	//Step 37-38: Read DC bus voltage (S-0-0380)
	37: //Step 37: Trigger FB
		_CmdReadDcBusVoltage( Execute := FALSE, Axis := _Axis );
		_CmdReadDcBusVoltage( Execute := TRUE, Timeout := DEFAULT_ADS_TIMEOUT, Axis := _Axis );
		IF _CmdReadDcBusVoltage.Busy THEN _Step := 38; END_IF
		
	38: //Step 38: Check for errors and write to diagnostic parameter
		_CmdReadDcBusVoltage( Execute := FALSE, Axis := _Axis );
		IF NOT _CmdReadDcBusVoltage.Busy THEN
			IF NOT _CmdReadDcBusVoltage.Error THEN
				_DcBusVoltage	:= _CmdReadDcBusVoltage.DcBusVoltage;
			ELSE
				Error 			:= TRUE;
				ErrorStep		:= _Step;
				AdsErrId		:= _CmdReadDcBusVoltage.AdsErrId;
				SercosErrId		:= _CmdReadDcBusVoltage.SercosErrId;
			END_IF
			_Step := 39;
		END_IF
		
	//Step 39-40: Read actual main voltage (P-0-0200)
	39: //Step 39: Trigger FB
		_CmdReadMainVoltage( Execute := FALSE, Axis := _Axis );
		_CmdReadMainVoltage( Execute := TRUE, Timeout := DEFAULT_ADS_TIMEOUT, Axis := _Axis );
		IF _CmdReadMainVoltage.Busy THEN _Step := 40; END_IF
		
	40: //Step 40: Check for errors and write to diagnostic parameter
		_CmdReadMainVoltage( Execute := FALSE, Axis := _Axis );
		IF NOT _CmdReadMainVoltage.Busy THEN
			IF NOT _CmdReadMainVoltage.Error THEN
				_ActMainPeakVoltage	:= _CmdReadMainVoltage.ActualMainVoltage;
				_ActMainRMSVoltage	:= _ActMainPeakVoltage/(SQRT(2));	
			ELSE
				Error 				:= TRUE;
				ErrorStep			:= _Step;
				ErrorStep			:= _Step;
				AdsErrId			:= _CmdReadMainVoltage.AdsErrId;
				SercosErrId			:= _CmdReadMainVoltage.SercosErrId;
			END_IF	
			_Step := 41;		
		END_IF
		
	//Step 41-42: Read Safety State (P-0-2002) and set state bool	
	41: //Step 41: Trigger FB
		_CmdSoERead( Execute := FALSE, Axis :=_Axis);	
		_CmdSoERead( Execute := TRUE, Idn := P_0_IDN + 2002, Element :=16#40, pDstBuf :=ADR(_SafetyOptionState), BufLen :=SIZEOF(_SafetyOptionState), Timeout := DEFAULT_ADS_TIMEOUT, Axis := _Axis);
		IF _CmdSoERead.Busy THEN _Step := 42; END_IF
		
	42: //Step 42: Check for errors and write to field parameter
		_CmdSoERead(Execute:= FALSE, Axis := _Axis);
		IF NOT _CmdSoERead.Busy THEN	
			IF NOT _CmdSoERead.Error THEN
				_SafetyStateBool	:= _SafetyOptionState.0;
			ELSE
				Error				:= TRUE;
				ErrorStep			:= _Step;
				AdsErrId			:= _CmdSoERead.AdsErrId;
				SercosErrId			:= _CmdSoERead.SercosErrId;
			END_IF
			_Step := 43;
		END_IF
	
	//Step 43-44: Read torque peak (P-0-0094)	
	43: //Step 43: Trigger FB
		_CmdSoERead( Execute := FALSE, Axis :=_Axis);	
		_CmdSoERead( Execute := TRUE, Idn := P_0_IDN + 92, Element :=16#40, pDstBuf :=ADR(_TorquePeak), BufLen :=SIZEOF(_TorquePeak), Timeout := DEFAULT_ADS_TIMEOUT, Axis := _Axis);
		IF _CmdSoERead.Busy THEN _Step := 44; END_IF
		
	44: //Step 44: Check for errors and write to field parameter
		_CmdSoERead(Execute:= FALSE, Axis := _Axis);
		IF NOT _CmdSoERead.Busy THEN	
			IF NOT _CmdSoERead.Error THEN
				;
			ELSE
				Error			:= TRUE;
				ErrorStep		:= _Step;
				AdsErrId		:= _CmdSoERead.AdsErrId;
				SercosErrId		:= _CmdSoERead.SercosErrId;
			END_IF
			_Step := 45;
		END_IF
		
	//Step 45-46: Read torque feedback percentage (S-0-0084)	
	45: //Step 45: Trigger FB	
		_CmdSoERead( Execute := FALSE, Axis :=_Axis);	
		_CmdSoERead( Execute := TRUE, Idn := S_0_IDNs + 84, Element :=16#40, pDstBuf :=ADR(_TorqueFeedbackPercent), BufLen :=SIZEOF(_TorqueFeedbackPercent), Timeout := DEFAULT_ADS_TIMEOUT, Axis := _Axis);
		IF _CmdSoERead.Busy THEN _Step := 46; END_IF
		
	46: //Step 46: Check for errors and write to field parameter after converting percentage of peak into current Nm
		//Note: In drive manager value read for parameter is real, when read in code however the value returned is an int. i.e. Torque peak - in DM = 6.0, returned from SOE read 6000, Torque % - in DM = 6.7 returned 67. (check date size in IDN description manual for 16 bit or 23 bit size.
		_CmdSoERead(Execute:= FALSE, Axis := _Axis);
		IF NOT _CmdSoERead.Busy THEN	
			IF NOT _CmdSoERead.Error THEN 
				_TorqueFeedback := (INT_TO_REAL(_TorqueFeedbackPercent)/10)*(DINT_TO_LREAL(_TorquePeak)/100000);
			ELSE
				Error			:= TRUE;
				ErrorStep		:= _Step;
				AdsErrId		:= _CmdSoERead.AdsErrId;
				SercosErrId		:= _CmdSoERead.SercosErrId;
			END_IF
			_Step := 47;
		END_IF

	//Step 47-48: Read motor break current (P-0-0064)
	47: //Step 37: Trigger FB
		_CmdSoERead( Execute := FALSE, Axis :=_Axis);	
		_CmdSoERead( Execute := TRUE, Idn := P_0_IDN + 64, Element :=16#40, pDstBuf :=ADR(_ActMotorBreakCurrentRead), BufLen :=SIZEOF(_ActMotorBreakCurrentRead), Timeout := DEFAULT_ADS_TIMEOUT, Axis := _Axis);
		IF _CmdSoERead.Busy THEN _Step := 48; END_IF
		
	48: //Step 48: Check for errors and write to status parameter
		_CmdSoERead(Execute:= FALSE, Axis := _Axis);
		IF NOT _CmdSoERead.Busy THEN	
			IF NOT _CmdSoERead.Error THEN
				_ActMotorBreakCurrent := INT_TO_REAL(_ActMotorBreakCurrentRead)/1000;
			ELSE
				Error			:= TRUE;
				ErrorStep		:= _Step;
				AdsErrId		:= _CmdSoERead.AdsErrId;
				SercosErrId		:= _CmdSoERead.SercosErrId;
			END_IF
			_Step := 49;	
		END_IF
	
	49: //Step 49: Calulate normal torque limit from peak
		_NormalTorqueLimitNm := (UINT_TO_REAL(_NormalTorqueLimit)/100) * (DINT_TO_LREAL(_TorquePeak)/1000);
		_Step := 50;
	
	// Step 50-51: Get motor peak force (P-0-0128)
	50: //Step 50: Trigger FB
		_CmdSoERead( Execute := FALSE, Axis :=_Axis);	
		_CmdSoERead( Execute := TRUE, Idn := P_0_IDN + 128, Element :=16#40, pDstBuf :=ADR(_MotorPeakForceRead), BufLen :=SIZEOF(_MotorPeakForceRead), Timeout := DEFAULT_ADS_TIMEOUT, Axis := _Axis);
		IF _CmdSoERead.Busy THEN _Step := 51; END_IF
		
	51: //Step 48: Check for errors and write to status parameter
		_CmdSoERead(Execute:= FALSE, Axis := _Axis);
		IF NOT _CmdSoERead.Busy THEN	
			IF NOT _CmdSoERead.Error THEN
				_MotorPeakForce := UINT_TO_REAL(_MotorPeakForceRead)/1000;
			ELSE
				Error			:= TRUE;
				ErrorStep		:= _Step;
				AdsErrId		:= _CmdSoERead.AdsErrId;
				SercosErrId		:= _CmdSoERead.SercosErrId;
			END_IF
			_Step		:= 0;	
		END_IF
		
	52: //Display diagnostics function error
		IF Error THEN
			;
		END_IF
END_CASE
END_METHOD

METHOD PRIVATE M_Homing
VAR_INPUT
END_VAR
VAR_INST
             	                			
	_HomingJogPos						: BOOL;	
	{attribute 'tc_no_symbol'}                	                			
	_CMD_Home							: MC_HOME;
	{attribute 'tc_no_symbol'}                	                			
	_CMD_SetPosition					: MC_SETPOSITION;
	{attribute 'tc_no_symbol'}                	                			
	_CMD_SoEAX5000SetPositionOffset		: FB_SoEAX5000SetPositionOffset;
	{attribute 'tc_no_symbol'}   
	_SoEAX5000SetPositionOffsetBusyLatch: BOOL;								//Due to no done bit for function this bit latched on busy then for use in detecting falling edge
	{attribute 'tc_no_symbol'}                	                			
	_CMD_SoEAX5000DeletePositionOffset	: FB_SoEAX5000DeletePositionOffset;
	{attribute 'tc_no_symbol'}                	                				
	_CMD_HomeJOG						: MC_JOG;
	{attribute 'tc_no_symbol'}                	                			
	_R_Trig								: ARRAY[0..6] OF R_TRIG;
END_VAR
// ----------------------------------------
// Homing Outputs
// ----------------------------------------
_HomingEN:=_CMD_Home.Busy OR _CMD_SetPosition.Busy OR _CMD_SoEAX5000SetPositionOffset.Busy;
IF _CMD_Home.Busy OR _CMD_SetPosition.Busy OR _CMD_SoEAX5000SetPositionOffset.Busy THEN _Homed := FALSE; END_IF
IF _CMD_Home.Done OR _CMD_SetPosition.Done OR _R_Trig[1].Q THEN _Homed := TRUE;_SoEAX5000SetPositionOffsetBusyLatch:=FALSE; END_IF

// ----------------------------------------
// Error Handler	
// ----------------------------------------
_r_Trig[0](clk :=
(_CMD_Home.Execute AND _CMD_Home.Error) OR 
(_CMD_SetPosition.Execute AND _CMD_SetPosition.Error) OR
(_CMD_SoEAX5000DeletePositionOffset.Execute AND _CMD_SoEAX5000DeletePositionOffset.Error) OR
(_CMD_SoEAX5000SetPositionOffset.Execute AND _CMD_SoEAX5000SetPositionOffset.Error));


// ----------------------------------------
// Manual Home Selection	
// ----------------------------------------
IF _ManHome.Select AND NOT _ManHome.Interlock THEN
	_ManHome.Select :=TRUE;
ELSE
	_ManHome.Select :=FALSE;
END_IF

IF ((_HomeMode < 3) AND NOT Control.PackMLState.Stopped AND NOT Control.PackMLState.Idle)  THEN
	_ManHome.Messages:= 'Axis Cannot be homed.$LSystem is not in an Stopped or Idle State.';
ELSIF((_HomeMode >= 3) AND NOT Control.PackMLState.Aborted) THEN
	_ManHome.Messages:= 'Axis Cannot be homed as the Machine is not De-energized.$LSystem is not in an Aborted State';
ELSIF _r_Trig[0].Q THEN
	_ManHome.Messages:= 'Axis Homing Error Occurred';
ELSE
	IF (_HomeMode < 3) THEN
		_ManHome.Messages:= 'Axis Ready to be Homed.$LThis will cause motion towards the Switch.';
	ELSE
		_ManHome.Messages:= 'Axis Ready to be Homed.$LThe Axis will remain stationary.';
	END_IF
END_IF


IF _CMD_Home.Done OR _CMD_SetPosition.Done OR _R_Trig[1].Q
	OR ((_HomeMode < 3) AND NOT Control.PackMLState.Stopped AND NOT Control.PackMLState.Idle)
	OR ((_HomeMode >= 3) AND NOT Control.PackMLState.Aborted)
	OR _r_Trig[0].Q THEN
	_ManHome.Interlock :=TRUE; 
ELSE
	_ManHome.Interlock :=FALSE;
END_IF


IF _ManHome.Select  THEN
	_ManHome.Queued :=TRUE;
	_ManHome.Messages:= 'Axis Homing Queued.';
ELSE
	_ManHome.Queued :=FALSE;
END_IF

IF _ManHome.Queued  THEN
	_ManHome.Messages:= 'Axis Homing in Progress.';
	_ManHome.Enabled :=TRUE;
ELSE
	_ManHome.Enabled :=FALSE;
END_IF

// ----------------------------------------
// MC Home	
// ----------------------------------------	
_CMD_Home(
	Axis:= _Axis, 
	Execute:= (_AutoHome OR _ManHome.Enabled) AND _HomeMode <=2,
	HomingMode:= MC_DefaultHoming, 
	BufferMode:= , 
	Options:= , 
	bCalibrationCam:= HomingInput, 
	Done=> , 
	Busy=> , 
	Active=> , 
	CommandAborted=> , 
	Error=> , 
	ErrorID=> );
_R_Trig[3](CLK:=_CMD_Home.Error);IF _R_Trig[3].Q THEN _AlarmNum := _CMD_Home.ErrorID; END_IF	

// ----------------------------------------
// MC Set Position	
// ----------------------------------------			
_CMD_SetPosition(
	Axis:= _Axis, 
	Execute:= (_AutoHome OR _ManHome.Enabled) AND _HomeMode = 3, 
	Position:= _PosMoveHome.Position, 
	Mode:= FALSE, 
	Options:= , 
	Done=> , 
	Busy=> , 
	Error=> , 
	ErrorID=> );	
_R_Trig[4](CLK:=_CMD_SetPosition.Error);IF _R_Trig[4].Q THEN _AlarmNum := _CMD_SetPosition.ErrorID; END_IF	

// ----------------------------------------
// MC Set Position Offset	
// ----------------------------------------		
//* Note to Set P-0-0275 = 2.Use Drive Memory	
_CMD_SoEAX5000SetPositionOffset(
	Execute:= (_AutoHome OR _ManHome.Enabled) AND _HomeMode = 4, 
	Position:= _PosMoveHome.Position, 
	Relative:= FALSE, 
	Feedback:= tc2_mc2_Drive.E_PositionOffsetFeedback.ePositionOffsetFeedback1, 
	Memory:=  tc2_mc2_Drive.E_PositionOffsetMemory.ePositionOffsetMemory_Drive, 
	Busy=> , 
	Error=> , 
	ErrorID=> , 
	Axis:= _Axis);
_R_Trig[5](CLK:=_CMD_SoEAX5000SetPositionOffset.Error);IF _R_Trig[5].Q THEN _AlarmNum := _CMD_SoEAX5000SetPositionOffset.ErrorID; END_IF
IF _CMD_SoEAX5000SetPositionOffset.Busy THEN _SoEAX5000SetPositionOffsetBusyLatch := TRUE; END_IF
_R_Trig[1](CLK:=_SoEAX5000SetPositionOffsetBusyLatch AND NOT _CMD_SoEAX5000SetPositionOffset.Busy);
END_METHOD

METHOD PRIVATE M_Jogging
VAR_INPUT
END_VAR
VAR_INST
	{attribute 'tc_no_symbol'}                	                			
	_accelRate							: LREAL;
	{attribute 'tc_no_symbol'}                	                			
	_decelRate							: LREAL;
	{attribute 'tc_no_symbol'}                	                			
	_jerkTime							: LREAL;
	{attribute 'tc_no_symbol'}                	                			
	_jerkValue							: LREAL;
	{attribute 'tc_no_symbol'}                	                			
	_enableJog							: BOOL;
	{attribute 'tc_no_symbol'}                	                			
	_enableManPos						: BOOL;
	{attribute 'tc_no_symbol'}                	                			
	_manPosAbsActive					: BOOL;
	{attribute 'tc_no_symbol'}                	                			
	_manPosModActive					: BOOL;
	{attribute 'tc_no_symbol'}                	                			
	_manPosRelActive					: BOOL;
	{attribute 'tc_no_symbol'}                	                			
	_CMD_JOG							: MC_JOG;
	{attribute 'tc_no_symbol'}                	                			
	_CMD_MovePosManAbs					: MC_MOVEABSOLUTE;
	{attribute 'tc_no_symbol'}                	                			
	_CMD_MovePosManMod					: MC_MOVEMODULO;
	{attribute 'tc_no_symbol'}                	                			
	_CMD_MovePosManRel					: MC_MOVERELATIVE;
	{attribute 'tc_no_symbol'}                	                			
	_CMD_ManMoveHalt					: MC_HALT;
END_VAR
VAR_INST // added by the converter: edge detectors and wires of the graphical bodies
    _w1, _w2 : BOOL;
    _rt1, _rt2, _rt3, _rt4, _rt5 : R_TRIG;
END_VAR
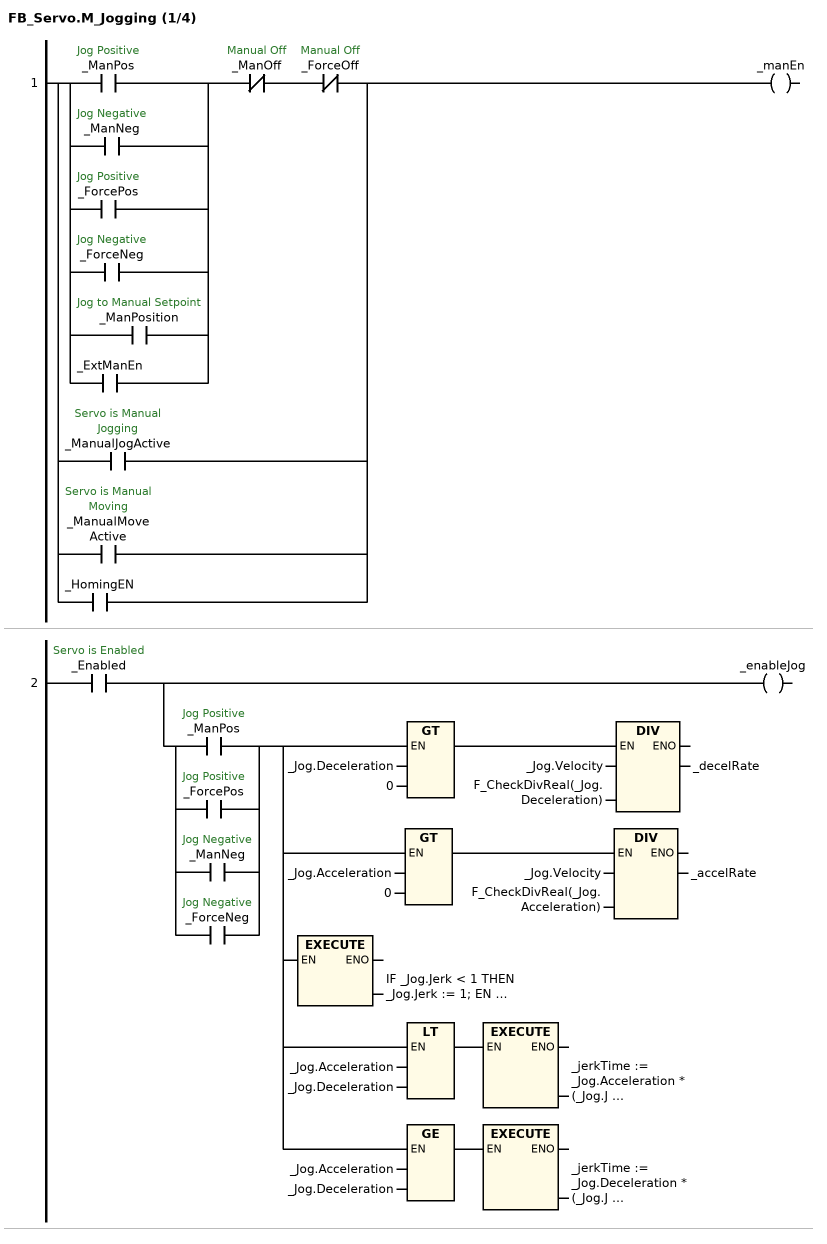
// NETWORK 1
//   _ManPos: Jog Positive
//   _ManNeg: Jog Negative
//   _ForcePos: Jog Positive
//   _ForceNeg: Jog Negative
//   _ManPosition: Jog to Manual Setpoint
//   _ManOff: Manual Off
//   _ForceOff: Manual Off
//   _ManualJogActive: Servo is Manual Jogging
//   _ManualMoveActive: Servo is Manual Moving
_manEn := (_ManPos OR _ManNeg OR _ForcePos OR _ForceNeg OR _ManPosition OR _ExtManEn) AND NOT _ManOff AND NOT _ForceOff OR _ManualJogActive OR _ManualMoveActive OR _HomingEN;

// NETWORK 2
//   _Enabled: Servo is Enabled
//   _ManPos: Jog Positive
//   _ForcePos: Jog Positive
//   _ManNeg: Jog Negative
//   _ForceNeg: Jog Negative
//   _Jog.Velocity: Velocity Value of Move
//   F_CheckDivReal(_Jog.Deceleration): Deceleration Value of Move
//   F_CheckDivReal(_Jog.Acceleration): Accleration Value of Move
//   _Jog.Acceleration: Accleration Value of Move
//   _Jog.Deceleration: Deceleration Value of Move
_enableJog := _Enabled;
_w1 := _Enabled AND (_ManPos OR _ForcePos OR _ManNeg OR _ForceNeg);
IF _w1 AND _Jog.Deceleration > 0 THEN _decelRate := _Jog.Velocity / (F_CheckDivReal(_Jog.Deceleration)); END_IF
IF _w1 AND _Jog.Acceleration > 0 THEN _accelRate := _Jog.Velocity / (F_CheckDivReal(_Jog.Acceleration)); END_IF
IF _w1 THEN
    IF _Jog.Jerk < 1 THEN _Jog.Jerk := 1; END_IF
    IF _Jog.Jerk > 100 THEN _Jog.Jerk := 100; END_IF
END_IF
IF _w1 AND _Jog.Acceleration < _Jog.Deceleration THEN
    _jerkTime := _Jog.Acceleration * (_Jog.Jerk / 100);
    IF _jerkTime > 0 THEN
    	_jerkValue := _accelRate / F_CheckDivReal(LREAL_TO_REAL(_jerkTime));
    END_IF
END_IF
IF _w1 AND _Jog.Acceleration >= _Jog.Deceleration THEN
    _jerkTime := _Jog.Deceleration * (_Jog.Jerk / 100);
    IF _jerkTime > 0 THEN
    	_jerkValue := _decelRate / F_CheckDivReal(LREAL_TO_REAL(_jerkTime));
    END_IF
END_IF

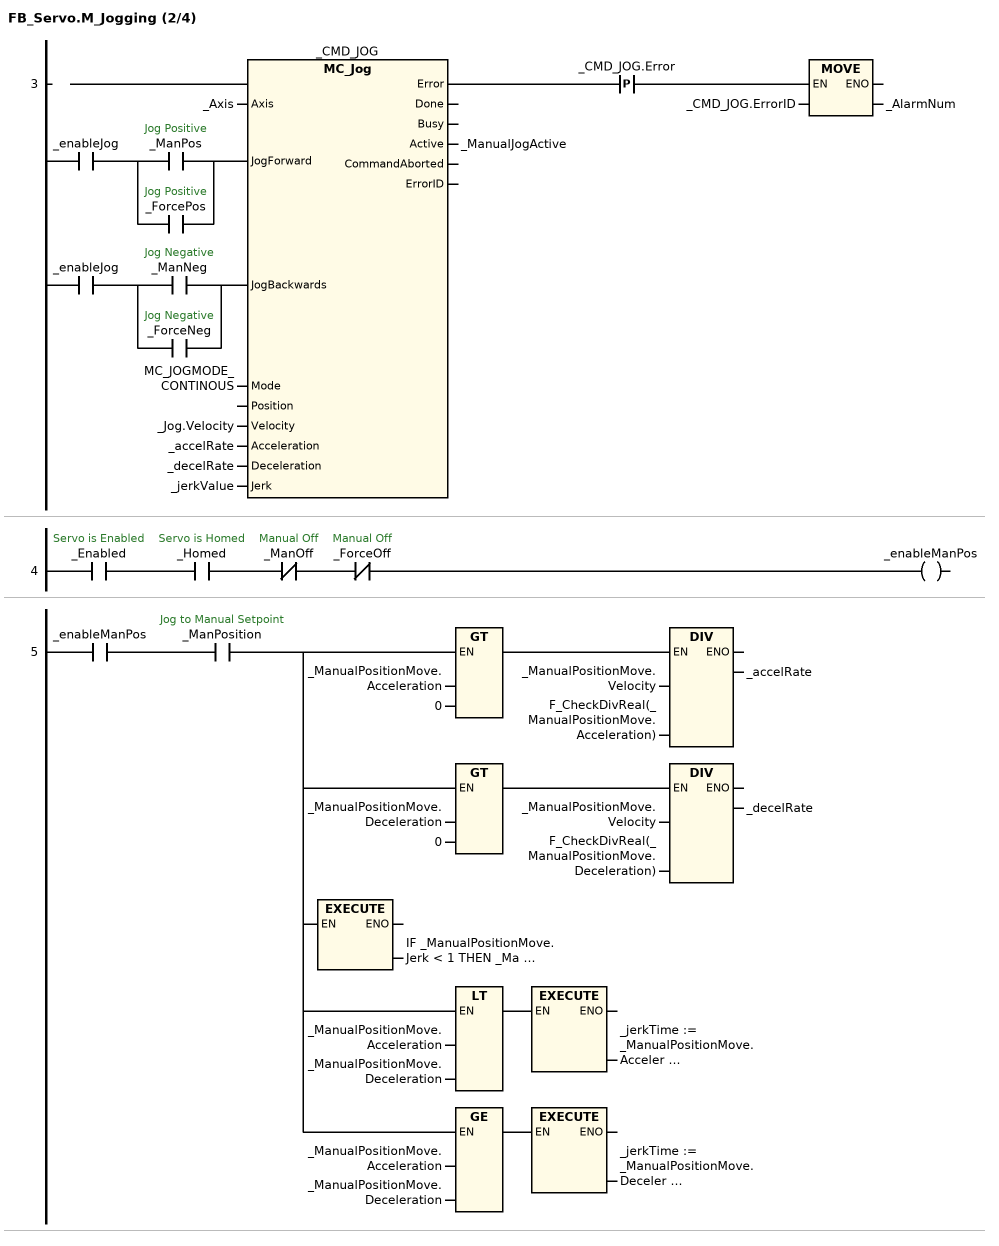
// NETWORK 3
//   _ManPos: Jog Positive
//   _ForcePos: Jog Positive
//   _ManNeg: Jog Negative
//   _ForceNeg: Jog Negative
//   MC_JOGMODE_CONTINOUS: axis moves as long as the jog button is pressed using parameterized dynamics
//   _Jog.Velocity: Velocity Value of Move
//   _ManualJogActive: Servo is Manual Jogging
_CMD_JOG(
    Axis := _Axis,
    JogForward := _enableJog AND (_ManPos OR _ForcePos),
    JogBackwards := _enableJog AND (_ManNeg OR _ForceNeg),
    Mode := MC_JOGMODE_CONTINOUS,
    Velocity := _Jog.Velocity,
    Acceleration := _accelRate,
    Deceleration := _decelRate,
    Jerk := _jerkValue,
    Active => _ManualJogActive); // MC_Jog
_rt1(CLK := _CMD_JOG.Error);
IF _CMD_JOG.Error AND _rt1.Q THEN _AlarmNum := _CMD_JOG.ErrorID; END_IF

// NETWORK 4
//   _Enabled: Servo is Enabled
//   _Homed: Servo is Homed
//   _ManOff: Manual Off
//   _ForceOff: Manual Off
_enableManPos := _Enabled AND _Homed AND NOT _ManOff AND NOT _ForceOff;

// NETWORK 5
//   _ManPosition: Jog to Manual Setpoint
//   _ManualPositionMove.Velocity: Velocity Value of Move
//   F_CheckDivReal(_ManualPositionMove.Acceleration): Accleration Value of Move
//   F_CheckDivReal(_ManualPositionMove.Deceleration): Deceleration Value of Move
//   _ManualPositionMove.Acceleration: Accleration Value of Move
//   _ManualPositionMove.Deceleration: Deceleration Value of Move
_w2 := _enableManPos AND _ManPosition;
IF _w2 AND _ManualPositionMove.Acceleration > 0 THEN
    _accelRate := _ManualPositionMove.Velocity / (F_CheckDivReal(_ManualPositionMove.Acceleration));
END_IF
IF _w2 AND _ManualPositionMove.Deceleration > 0 THEN
    _decelRate := _ManualPositionMove.Velocity / (F_CheckDivReal(_ManualPositionMove.Deceleration));
END_IF
IF _w2 THEN
    IF _ManualPositionMove.Jerk < 1 THEN _ManualPositionMove.Jerk := 1; END_IF
    IF _ManualPositionMove.Jerk > 100 THEN _ManualPositionMove.Jerk := 100; END_IF
END_IF
IF _w2 AND _ManualPositionMove.Acceleration < _ManualPositionMove.Deceleration THEN
    _jerkTime := _ManualPositionMove.Acceleration * (_ManualPositionMove.Jerk / 100);
    IF _jerkTime > 0 THEN
    	_jerkValue := _accelRate / F_CheckDivReal(LREAL_TO_REAL(_jerkTime));
    END_IF
END_IF
IF _w2 AND _ManualPositionMove.Acceleration >= _ManualPositionMove.Deceleration THEN
    _jerkTime := _ManualPositionMove.Deceleration * (_ManualPositionMove.Jerk / 100);
    IF _jerkTime > 0 THEN
    	_jerkValue := _decelRate / F_CheckDivReal(LREAL_TO_REAL(_jerkTime));
    END_IF
END_IF

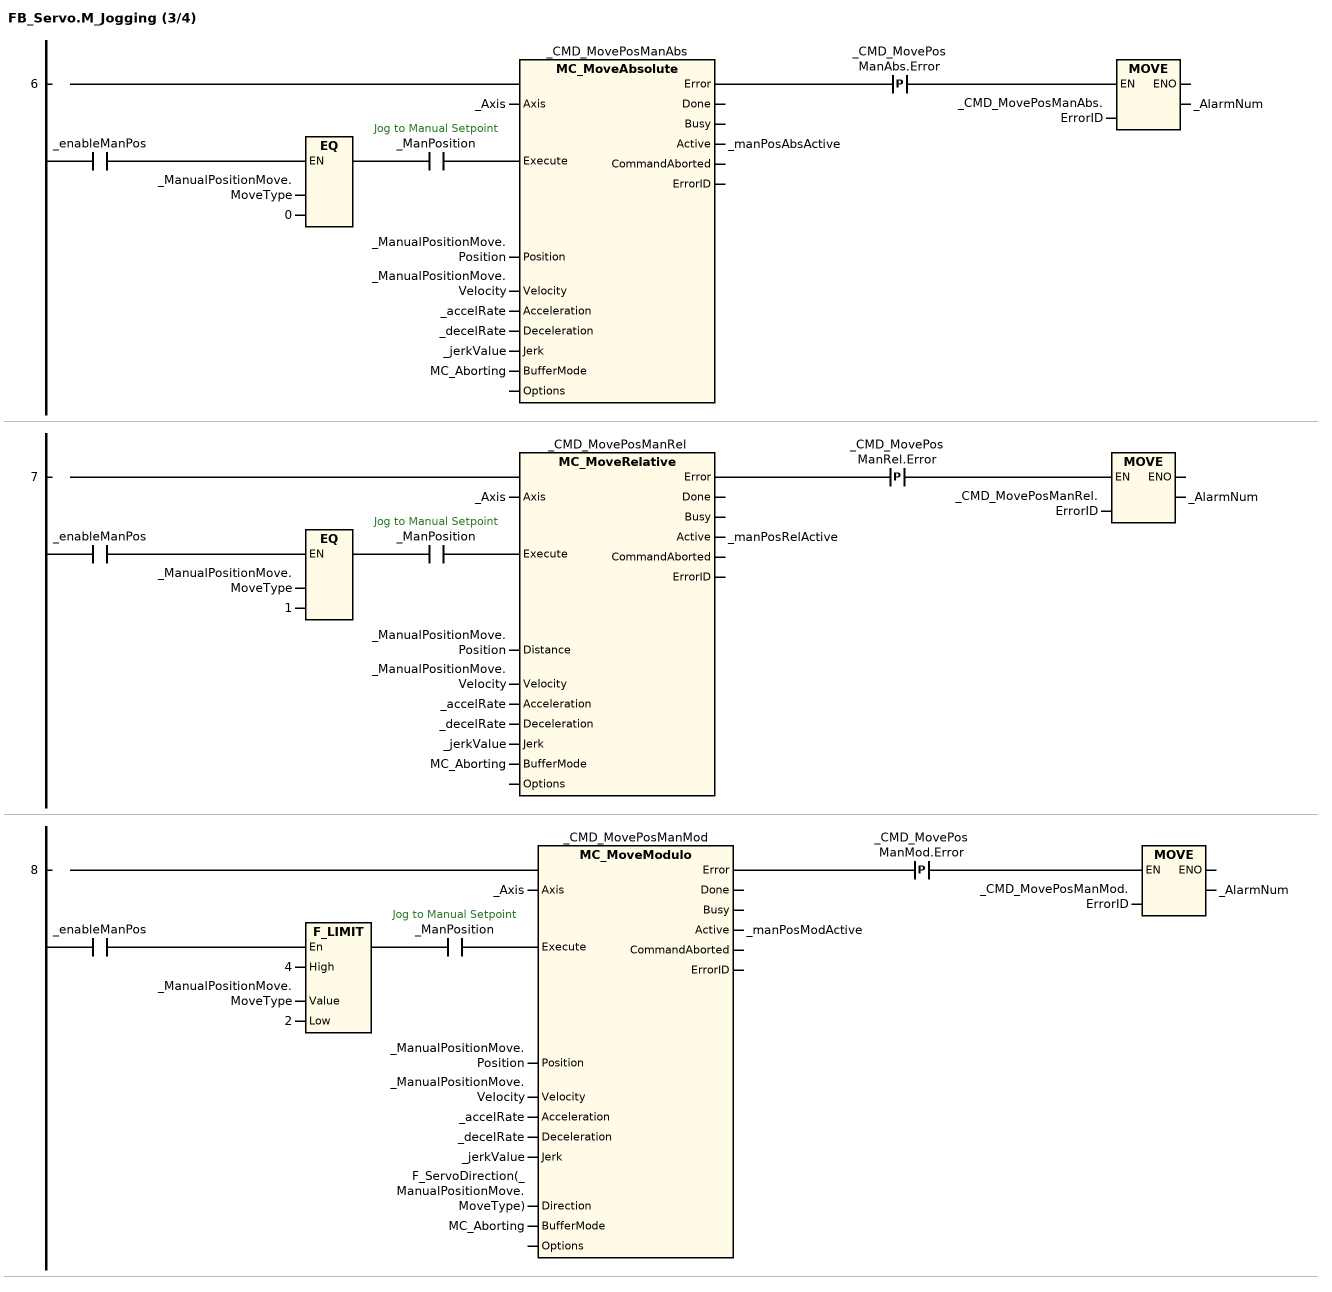
// NETWORK 6
//   _ManualPositionMove.MoveType: Move Type Configuration of Positional Move
//   _ManPosition: Jog to Manual Setpoint
//   _ManualPositionMove.Position: Position Value to Move to
//   _ManualPositionMove.Velocity: Velocity Value of Move
_CMD_MovePosManAbs(
    Axis := _Axis,
    Execute := (_enableManPos AND _ManualPositionMove.MoveType = 0) AND _ManPosition,
    Position := _ManualPositionMove.Position,
    Velocity := _ManualPositionMove.Velocity,
    Acceleration := _accelRate,
    Deceleration := _decelRate,
    Jerk := _jerkValue,
    BufferMode := MC_Aborting,
    Active => _manPosAbsActive); // MC_MoveAbsolute
_rt2(CLK := _CMD_MovePosManAbs.Error);
IF _CMD_MovePosManAbs.Error AND _rt2.Q THEN _AlarmNum := _CMD_MovePosManAbs.ErrorID; END_IF

// NETWORK 7
//   _ManualPositionMove.MoveType: Move Type Configuration of Positional Move
//   _ManPosition: Jog to Manual Setpoint
//   _ManualPositionMove.Position: Position Value to Move to
//   _ManualPositionMove.Velocity: Velocity Value of Move
_CMD_MovePosManRel(
    Axis := _Axis,
    Execute := (_enableManPos AND _ManualPositionMove.MoveType = 1) AND _ManPosition,
    Distance := _ManualPositionMove.Position,
    Velocity := _ManualPositionMove.Velocity,
    Acceleration := _accelRate,
    Deceleration := _decelRate,
    Jerk := _jerkValue,
    BufferMode := MC_Aborting,
    Active => _manPosRelActive); // MC_MoveRelative
_rt3(CLK := _CMD_MovePosManRel.Error);
IF _CMD_MovePosManRel.Error AND _rt3.Q THEN _AlarmNum := _CMD_MovePosManRel.ErrorID; END_IF

// NETWORK 8
//   _ManualPositionMove.MoveType: Move Type Configuration of Positional Move
//   _ManPosition: Jog to Manual Setpoint
//   _ManualPositionMove.Position: Position Value to Move to
//   _ManualPositionMove.Velocity: Velocity Value of Move
_CMD_MovePosManMod(
    Axis := _Axis,
    Execute := F_LIMIT(En := _enableManPos, High := 4, Value := _ManualPositionMove.MoveType, Low := 2) AND _ManPosition,
    Position := _ManualPositionMove.Position,
    Velocity := _ManualPositionMove.Velocity,
    Acceleration := _accelRate,
    Deceleration := _decelRate,
    Jerk := _jerkValue,
    Direction := F_ServoDirection(_ManualPositionMove.MoveType),
    BufferMode := MC_Aborting,
    Active => _manPosModActive); // MC_MoveModulo
_rt4(CLK := _CMD_MovePosManMod.Error);
IF _CMD_MovePosManMod.Error AND _rt4.Q THEN _AlarmNum := _CMD_MovePosManMod.ErrorID; END_IF

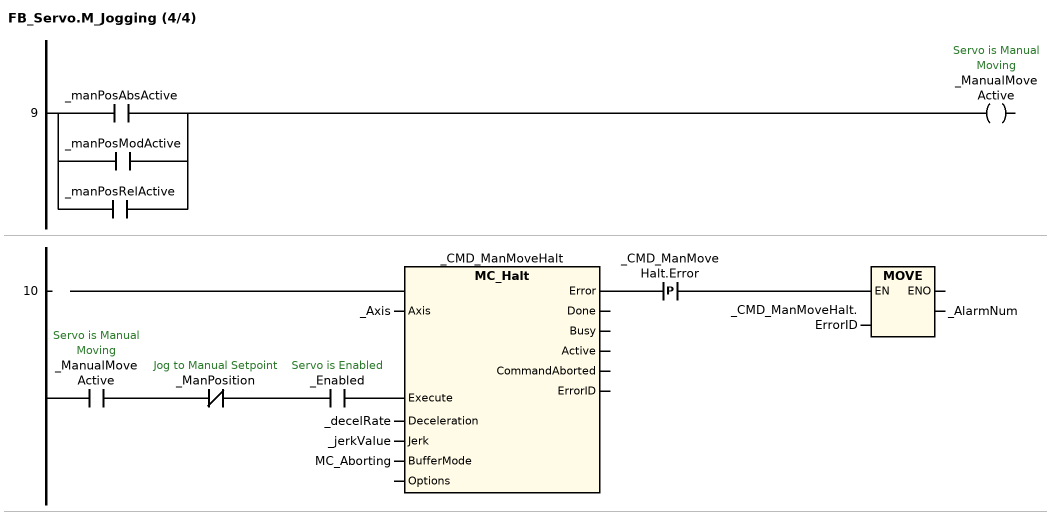
// NETWORK 9
//   _ManualMoveActive: Servo is Manual Moving
_ManualMoveActive := _manPosAbsActive OR _manPosModActive OR _manPosRelActive;

// NETWORK 10
//   _ManualMoveActive: Servo is Manual Moving
//   _ManPosition: Jog to Manual Setpoint
//   _Enabled: Servo is Enabled
_CMD_ManMoveHalt(
    Axis := _Axis,
    Execute := _ManualMoveActive AND NOT _ManPosition AND _Enabled,
    Deceleration := _decelRate,
    Jerk := _jerkValue,
    BufferMode := MC_Aborting); // MC_Halt
_rt5(CLK := _CMD_ManMoveHalt.Error);
IF _CMD_ManMoveHalt.Error AND _rt5.Q THEN _AlarmNum := _CMD_ManMoveHalt.ErrorID; END_IF
END_METHOD

METHOD PRIVATE M_MotionDynamicMove
VAR_INPUT
END_VAR
VAR_INST
	{attribute 'tc_no_symbol'}                	                			
	_fb_MovePosDynamic			: ARRAY [1..4] OF FB_ServoMotionDynamics;
	{attribute 'tc_no_symbol'}                	                			
	_enableDynamicMove			: BOOL;
	{attribute 'tc_no_symbol'}                	                			
	_Pos2MoveStart				: ST_MovePosition_SP;
	{attribute 'tc_no_symbol'}                	                			
	_CMD_MoveDynamicAbsStart	: ARRAY[1..4] OF MC_MOVEABSOLUTE;
	{attribute 'tc_no_symbol'}                	                			
	_CMD_MoveDynamicAbsEnd		: ARRAY[1..4] OF MC_MOVEABSOLUTE;
END_VAR
VAR_INST // added by the converter: edge detectors and wires of the graphical bodies
    _rt1, _rt2, _rt3, _rt4, _rt5, _rt6, _rt7, _rt8, _rt9, _rt10 : R_TRIG;
    _w1, _w2 : BOOL;
END_VAR
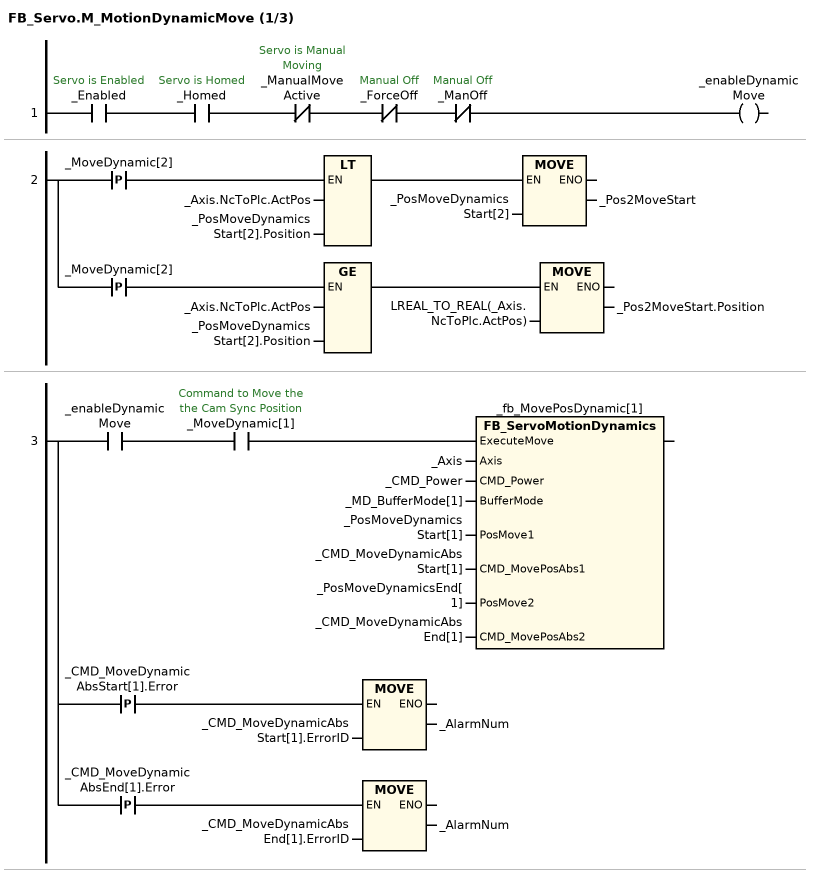
// NETWORK 1
//   _Enabled: Servo is Enabled
//   _Homed: Servo is Homed
//   _ManualMoveActive: Servo is Manual Moving
//   _ForceOff: Manual Off
//   _ManOff: Manual Off
_enableDynamicMove := _Enabled AND _Homed AND NOT _ManualMoveActive AND NOT _ForceOff AND NOT _ManOff;

// NETWORK 2
_rt1(CLK := _MoveDynamic[2]);
_w1 := _rt1.Q AND _Axis.NcToPlc.ActPos < _PosMoveDynamicsStart[2].Position;
IF _w1 THEN _Pos2MoveStart := _PosMoveDynamicsStart[2]; END_IF
_rt2(CLK := _MoveDynamic[2]);
_w2 := _rt2.Q AND _Axis.NcToPlc.ActPos >= _PosMoveDynamicsStart[2].Position;
IF _w2 THEN _Pos2MoveStart.Position := LREAL_TO_REAL(_Axis.NcToPlc.ActPos); END_IF

// NETWORK 3
//   _MoveDynamic[1]: Command to Move the the Cam Sync Position
_fb_MovePosDynamic[1](
    ExecuteMove := _enableDynamicMove AND _MoveDynamic[1],
    Axis := _Axis,
    CMD_Power := _CMD_Power,
    BufferMode := _MD_BufferMode[1],
    PosMove1 := _PosMoveDynamicsStart[1],
    CMD_MovePosAbs1 := _CMD_MoveDynamicAbsStart[1],
    PosMove2 := _PosMoveDynamicsEnd[1],
    CMD_MovePosAbs2 := _CMD_MoveDynamicAbsEnd[1]); // FB_ServoMotionDynamics
_rt3(CLK := _CMD_MoveDynamicAbsStart[1].Error);
IF _rt3.Q THEN _AlarmNum := _CMD_MoveDynamicAbsStart[1].ErrorID; END_IF
_rt4(CLK := _CMD_MoveDynamicAbsEnd[1].Error);
IF _rt4.Q THEN _AlarmNum := _CMD_MoveDynamicAbsEnd[1].ErrorID; END_IF

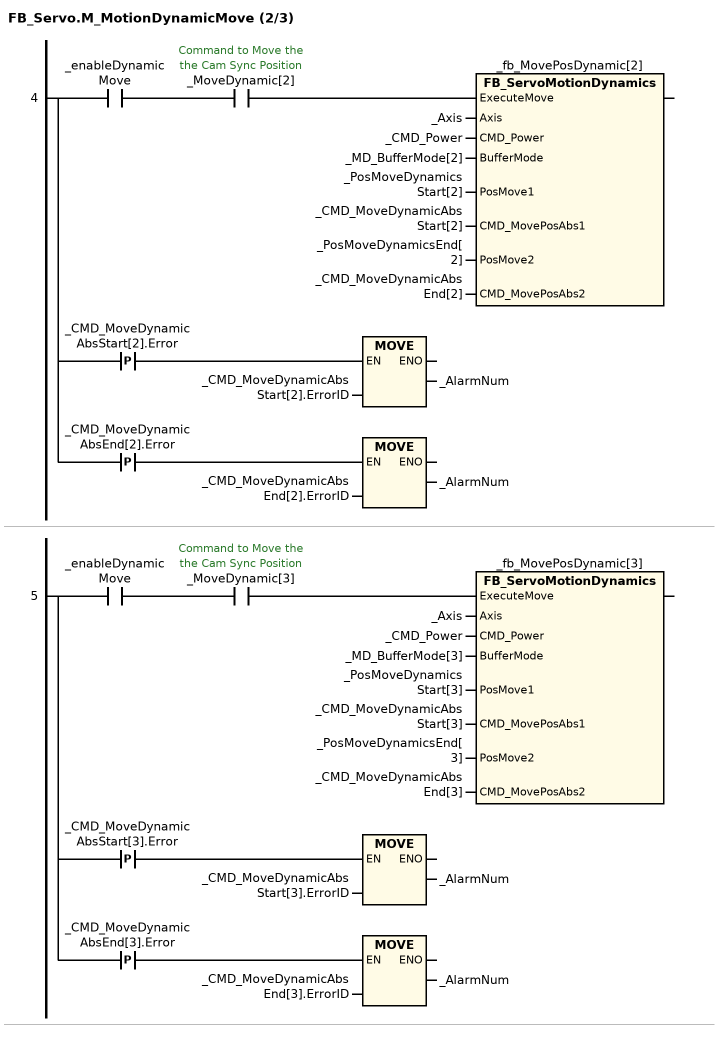
// NETWORK 4
//   _MoveDynamic[2]: Command to Move the the Cam Sync Position
_fb_MovePosDynamic[2](
    ExecuteMove := _enableDynamicMove AND _MoveDynamic[2],
    Axis := _Axis,
    CMD_Power := _CMD_Power,
    BufferMode := _MD_BufferMode[2],
    PosMove1 := _PosMoveDynamicsStart[2],
    CMD_MovePosAbs1 := _CMD_MoveDynamicAbsStart[2],
    PosMove2 := _PosMoveDynamicsEnd[2],
    CMD_MovePosAbs2 := _CMD_MoveDynamicAbsEnd[2]); // FB_ServoMotionDynamics
_rt5(CLK := _CMD_MoveDynamicAbsStart[2].Error);
IF _rt5.Q THEN _AlarmNum := _CMD_MoveDynamicAbsStart[2].ErrorID; END_IF
_rt6(CLK := _CMD_MoveDynamicAbsEnd[2].Error);
IF _rt6.Q THEN _AlarmNum := _CMD_MoveDynamicAbsEnd[2].ErrorID; END_IF

// NETWORK 5
//   _MoveDynamic[3]: Command to Move the the Cam Sync Position
_fb_MovePosDynamic[3](
    ExecuteMove := _enableDynamicMove AND _MoveDynamic[3],
    Axis := _Axis,
    CMD_Power := _CMD_Power,
    BufferMode := _MD_BufferMode[3],
    PosMove1 := _PosMoveDynamicsStart[3],
    CMD_MovePosAbs1 := _CMD_MoveDynamicAbsStart[3],
    PosMove2 := _PosMoveDynamicsEnd[3],
    CMD_MovePosAbs2 := _CMD_MoveDynamicAbsEnd[3]); // FB_ServoMotionDynamics
_rt7(CLK := _CMD_MoveDynamicAbsStart[3].Error);
IF _rt7.Q THEN _AlarmNum := _CMD_MoveDynamicAbsStart[3].ErrorID; END_IF
_rt8(CLK := _CMD_MoveDynamicAbsEnd[3].Error);
IF _rt8.Q THEN _AlarmNum := _CMD_MoveDynamicAbsEnd[3].ErrorID; END_IF

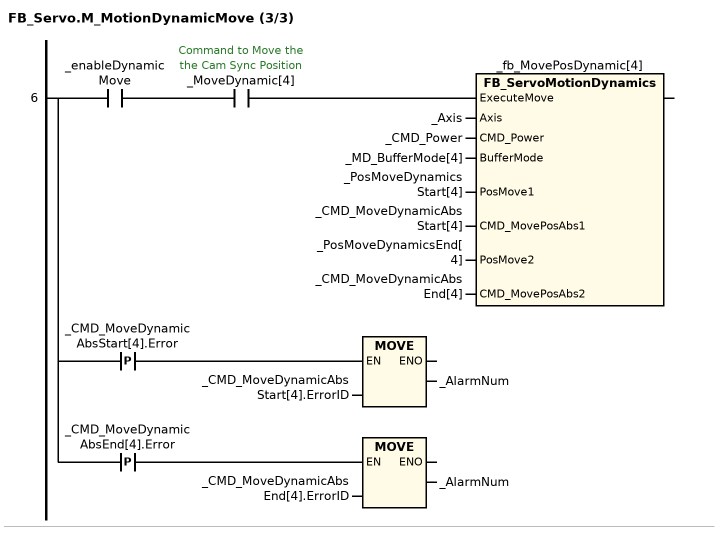
// NETWORK 6
//   _MoveDynamic[4]: Command to Move the the Cam Sync Position
_fb_MovePosDynamic[4](
    ExecuteMove := _enableDynamicMove AND _MoveDynamic[4],
    Axis := _Axis,
    CMD_Power := _CMD_Power,
    BufferMode := _MD_BufferMode[4],
    PosMove1 := _PosMoveDynamicsStart[4],
    CMD_MovePosAbs1 := _CMD_MoveDynamicAbsStart[4],
    PosMove2 := _PosMoveDynamicsEnd[4],
    CMD_MovePosAbs2 := _CMD_MoveDynamicAbsEnd[4]); // FB_ServoMotionDynamics
_rt9(CLK := _CMD_MoveDynamicAbsStart[4].Error);
IF _rt9.Q THEN _AlarmNum := _CMD_MoveDynamicAbsStart[4].ErrorID; END_IF
_rt10(CLK := _CMD_MoveDynamicAbsEnd[4].Error);
IF _rt10.Q THEN _AlarmNum := _CMD_MoveDynamicAbsEnd[4].ErrorID; END_IF
END_METHOD

METHOD PRIVATE M_MoveSuperImposed
VAR_INPUT
END_VAR
VAR_INST
	{attribute 'tc_no_symbol'}                	                			
	_enableSuperImposed					: BOOL;
	{attribute 'tc_no_symbol'}                	                			
	_CMD_MoveSuperImposed				: MC_MOVESUPERIMPOSED;
END_VAR
VAR_INST // added by the converter: edge detectors and wires of the graphical bodies
    _rt1 : R_TRIG;
END_VAR
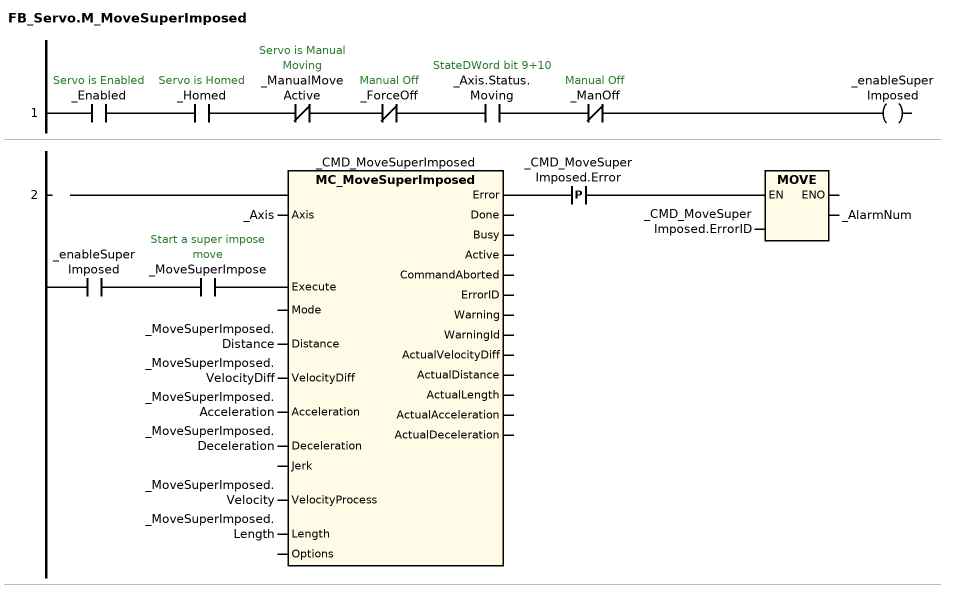
// NETWORK 1
//   _Enabled: Servo is Enabled
//   _Homed: Servo is Homed
//   _ManualMoveActive: Servo is Manual Moving
//   _ForceOff: Manual Off
//   _Axis.Status.Moving: StateDWord bit 9+10
//   _ManOff: Manual Off
_enableSuperImposed := _Enabled AND _Homed AND NOT _ManualMoveActive AND NOT _ForceOff AND _Axis.Status.Moving AND NOT _ManOff;

// NETWORK 2
//   _MoveSuperImpose: Start a super impose move
//   _MoveSuperImposed.Distance: Relative distance to catch up or fall back with the super imposed move
//   _MoveSuperImposed.VelocityDiff: Velocity Value of the catch up or fall back distance
//   _MoveSuperImposed.Acceleration: Accleration Value of Move
//   _MoveSuperImposed.Deceleration: Deceleration Value of Move
//   _MoveSuperImposed.Velocity: Velocity Value of Move without move super imposed
//   _MoveSuperImposed.Length: Length of the total move distance
_CMD_MoveSuperImposed(
    Axis := _Axis,
    Execute := _enableSuperImposed AND _MoveSuperImpose,
    Distance := _MoveSuperImposed.Distance,
    VelocityDiff := _MoveSuperImposed.VelocityDiff,
    Acceleration := _MoveSuperImposed.Acceleration,
    Deceleration := _MoveSuperImposed.Deceleration,
    VelocityProcess := _MoveSuperImposed.Velocity,
    Length := _MoveSuperImposed.Length); // MC_MoveSuperImposed
_rt1(CLK := _CMD_MoveSuperImposed.Error);
IF _CMD_MoveSuperImposed.Error AND _rt1.Q THEN _AlarmNum := _CMD_MoveSuperImposed.ErrorID; END_IF
END_METHOD

METHOD PRIVATE M_MoveToPosition
VAR_INPUT
END_VAR
VAR_INST
	{attribute 'tc_no_symbol'}                	                			
	_fb_MovePos							: ARRAY [1..4] OF FB_ServoMove;
	{attribute 'tc_no_symbol'}                	                			
	_fb_MovePosSync						: FB_ServoMove;
	{attribute 'tc_no_symbol'}                	                			
	_enableMove							: BOOL;
	{attribute 'tc_no_symbol'}                	                			
	_enableMoveHalt						: BOOL;
	{attribute 'tc_no_symbol'}                	                			
	_decelRateMoveHalt					: LREAL;
	{attribute 'tc_no_symbol'}                	                			
	_CMD_MovePosSyncAbs					: MC_MOVEABSOLUTE;
	{attribute 'tc_no_symbol'}                	                			
	_CMD_MovePosSyncMod					: MC_MOVEMODULO;
	{attribute 'tc_no_symbol'}                	                			
	_CMD_MovePosSyncRel					: MC_MOVERELATIVE;
	{attribute 'tc_no_symbol'}                	                			
	_CMD_MoveHalt						: MC_HALT;
	{attribute 'tc_no_symbol'}                	                			
	_CMD_MovePosAbs						: ARRAY[1..4] OF MC_MOVEABSOLUTE;
	{attribute 'tc_no_symbol'}                	                			
	_CMD_MovePosMod						: ARRAY[1..4] OF MC_MOVEMODULO;
	{attribute 'tc_no_symbol'}                	                			
	_CMD_MovePosRel						: ARRAY[1..4] OF MC_MOVERELATIVE;
	{attribute 'tc_no_symbol'}                	                			
	_R_Trig								: ARRAY[0..3] OF R_TRIG;
END_VAR
VAR_INST // added by the converter: edge detectors and wires of the graphical bodies
    _rt1, _rt2, _rt3, _rt4, _rt5, _rt6, _rt7, _rt8, _rt9, _rt10, _rt11, _rt12, _rt13, _rt14, _rt15, _rt16 : R_TRIG;
END_VAR
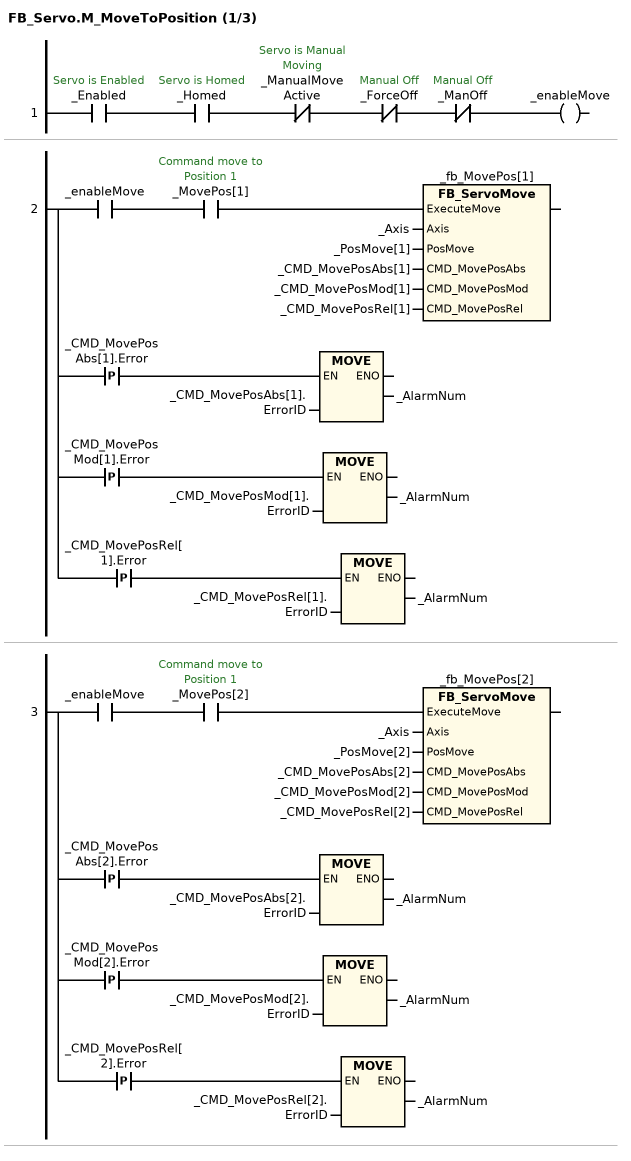
// NETWORK 1
//   _Enabled: Servo is Enabled
//   _Homed: Servo is Homed
//   _ManualMoveActive: Servo is Manual Moving
//   _ForceOff: Manual Off
//   _ManOff: Manual Off
_enableMove := _Enabled AND _Homed AND NOT _ManualMoveActive AND NOT _ForceOff AND NOT _ManOff;

// NETWORK 2
//   _MovePos[1]: Command move to Position 1
//   _PosMove[1]: Position 1 Move Setpoints
_fb_MovePos[1](
    ExecuteMove := _enableMove AND _MovePos[1],
    Axis := _Axis,
    PosMove := _PosMove[1],
    CMD_MovePosAbs := _CMD_MovePosAbs[1],
    CMD_MovePosMod := _CMD_MovePosMod[1],
    CMD_MovePosRel := _CMD_MovePosRel[1]); // FB_ServoMove
_rt1(CLK := _CMD_MovePosAbs[1].Error);
IF _rt1.Q THEN _AlarmNum := _CMD_MovePosAbs[1].ErrorID; END_IF
_rt2(CLK := _CMD_MovePosMod[1].Error);
IF _rt2.Q THEN _AlarmNum := _CMD_MovePosMod[1].ErrorID; END_IF
_rt3(CLK := _CMD_MovePosRel[1].Error);
IF _rt3.Q THEN _AlarmNum := _CMD_MovePosRel[1].ErrorID; END_IF

// NETWORK 3
//   _MovePos[2]: Command move to Position 1
//   _PosMove[2]: Position 1 Move Setpoints
_fb_MovePos[2](
    ExecuteMove := _enableMove AND _MovePos[2],
    Axis := _Axis,
    PosMove := _PosMove[2],
    CMD_MovePosAbs := _CMD_MovePosAbs[2],
    CMD_MovePosMod := _CMD_MovePosMod[2],
    CMD_MovePosRel := _CMD_MovePosRel[2]); // FB_ServoMove
_rt4(CLK := _CMD_MovePosAbs[2].Error);
IF _rt4.Q THEN _AlarmNum := _CMD_MovePosAbs[2].ErrorID; END_IF
_rt5(CLK := _CMD_MovePosMod[2].Error);
IF _rt5.Q THEN _AlarmNum := _CMD_MovePosMod[2].ErrorID; END_IF
_rt6(CLK := _CMD_MovePosRel[2].Error);
IF _rt6.Q THEN _AlarmNum := _CMD_MovePosRel[2].ErrorID; END_IF

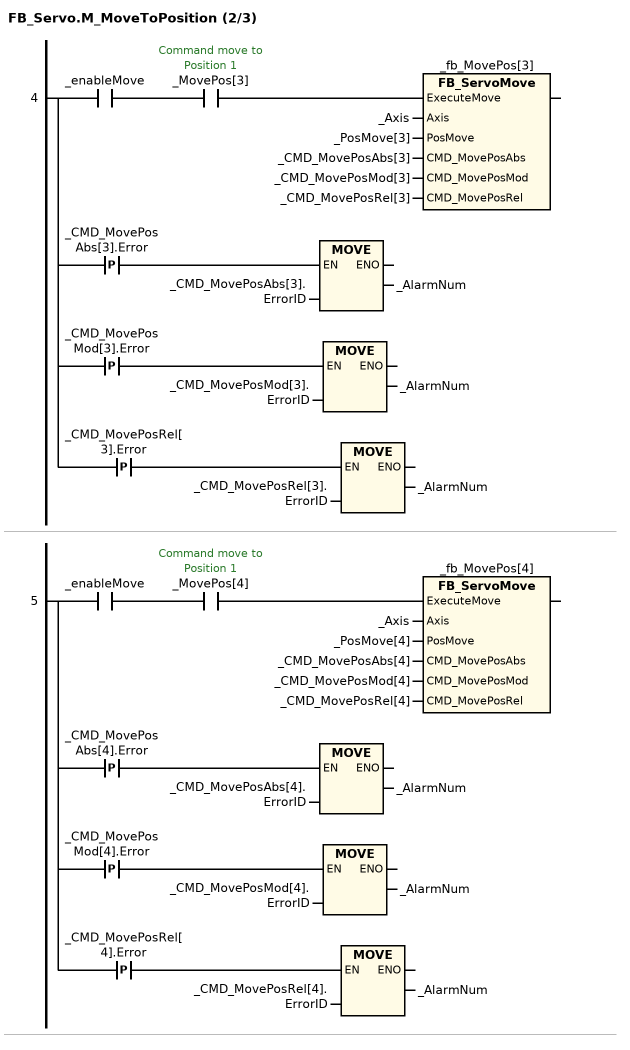
// NETWORK 4
//   _MovePos[3]: Command move to Position 1
//   _PosMove[3]: Position 1 Move Setpoints
_fb_MovePos[3](
    ExecuteMove := _enableMove AND _MovePos[3],
    Axis := _Axis,
    PosMove := _PosMove[3],
    CMD_MovePosAbs := _CMD_MovePosAbs[3],
    CMD_MovePosMod := _CMD_MovePosMod[3],
    CMD_MovePosRel := _CMD_MovePosRel[3]); // FB_ServoMove
_rt7(CLK := _CMD_MovePosAbs[3].Error);
IF _rt7.Q THEN _AlarmNum := _CMD_MovePosAbs[3].ErrorID; END_IF
_rt8(CLK := _CMD_MovePosMod[3].Error);
IF _rt8.Q THEN _AlarmNum := _CMD_MovePosMod[3].ErrorID; END_IF
_rt9(CLK := _CMD_MovePosRel[3].Error);
IF _rt9.Q THEN _AlarmNum := _CMD_MovePosRel[3].ErrorID; END_IF

// NETWORK 5
//   _MovePos[4]: Command move to Position 1
//   _PosMove[4]: Position 1 Move Setpoints
_fb_MovePos[4](
    ExecuteMove := _enableMove AND _MovePos[4],
    Axis := _Axis,
    PosMove := _PosMove[4],
    CMD_MovePosAbs := _CMD_MovePosAbs[4],
    CMD_MovePosMod := _CMD_MovePosMod[4],
    CMD_MovePosRel := _CMD_MovePosRel[4]); // FB_ServoMove
_rt10(CLK := _CMD_MovePosAbs[4].Error);
IF _rt10.Q THEN _AlarmNum := _CMD_MovePosAbs[4].ErrorID; END_IF
_rt11(CLK := _CMD_MovePosMod[4].Error);
IF _rt11.Q THEN _AlarmNum := _CMD_MovePosMod[4].ErrorID; END_IF
_rt12(CLK := _CMD_MovePosRel[4].Error);
IF _rt12.Q THEN _AlarmNum := _CMD_MovePosRel[4].ErrorID; END_IF

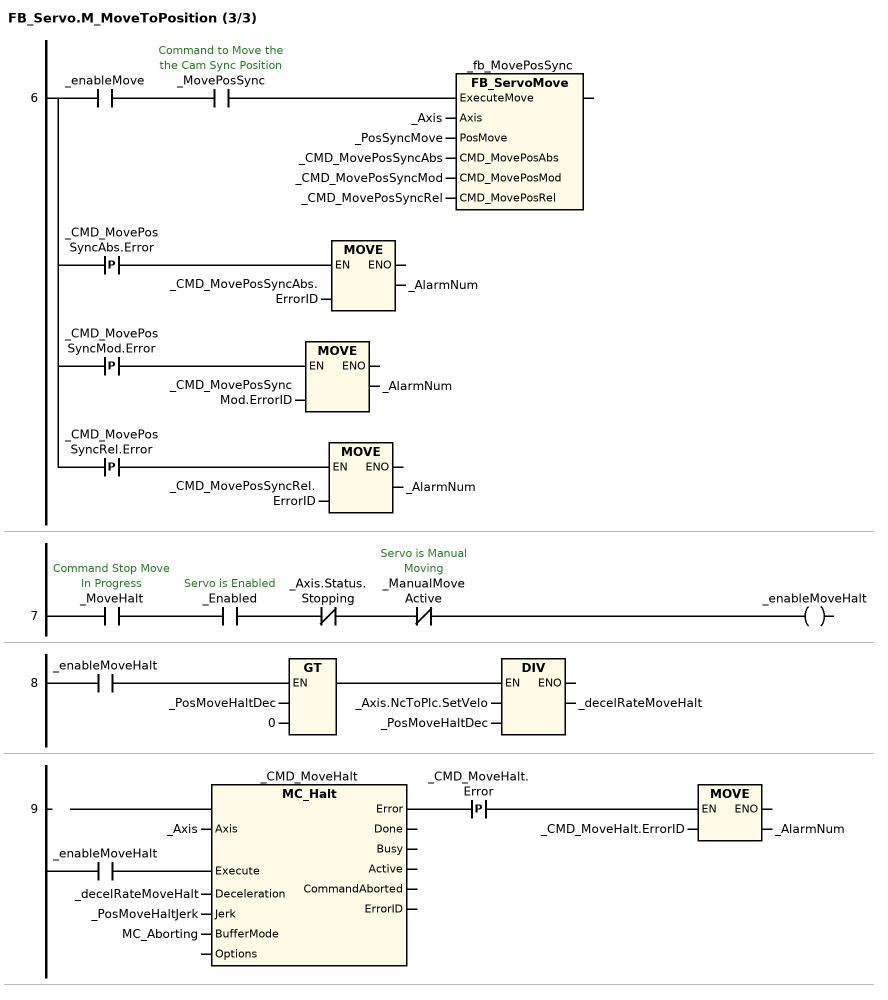
// NETWORK 6
//   _MovePosSync: Command to Move the the Cam Sync Position
//   _PosSyncMove: Sync Position Move Setpoints
_fb_MovePosSync(
    ExecuteMove := _enableMove AND _MovePosSync,
    Axis := _Axis,
    PosMove := _PosSyncMove,
    CMD_MovePosAbs := _CMD_MovePosSyncAbs,
    CMD_MovePosMod := _CMD_MovePosSyncMod,
    CMD_MovePosRel := _CMD_MovePosSyncRel); // FB_ServoMove
_rt13(CLK := _CMD_MovePosSyncAbs.Error);
IF _rt13.Q THEN _AlarmNum := _CMD_MovePosSyncAbs.ErrorID; END_IF
_rt14(CLK := _CMD_MovePosSyncMod.Error);
IF _rt14.Q THEN _AlarmNum := _CMD_MovePosSyncMod.ErrorID; END_IF
_rt15(CLK := _CMD_MovePosSyncRel.Error);
IF _rt15.Q THEN _AlarmNum := _CMD_MovePosSyncRel.ErrorID; END_IF

// NETWORK 7
//   _MoveHalt: Command Stop Move In Progress
//   _Enabled: Servo is Enabled
//   _ManualMoveActive: Servo is Manual Moving
_enableMoveHalt := _MoveHalt AND _Enabled AND NOT _Axis.Status.Stopping AND NOT _ManualMoveActive;

// NETWORK 8
//   _PosMoveHaltDec: Positional Move Halt Deceration
IF _enableMoveHalt AND _PosMoveHaltDec > 0 THEN
    _decelRateMoveHalt := _Axis.NcToPlc.SetVelo / _PosMoveHaltDec;
END_IF

// NETWORK 9
//   _PosMoveHaltJerk: Positional Move Halt Jerk
_CMD_MoveHalt(
    Axis := _Axis,
    Execute := _enableMoveHalt,
    Deceleration := _decelRateMoveHalt,
    Jerk := _PosMoveHaltJerk,
    BufferMode := MC_Aborting); // MC_Halt
_rt16(CLK := _CMD_MoveHalt.Error);
IF _CMD_MoveHalt.Error AND _rt16.Q THEN _AlarmNum := _CMD_MoveHalt.ErrorID; END_IF
END_METHOD

METHOD PRIVATE M_SettingsControl
VAR_INPUT
END_VAR
VAR_INST
	{attribute 'tc_no_symbol'}                	                			
	_homeOffsetPosition_Used			: LREAL;
	{attribute 'tc_no_symbol'}                	                			
	_maxPositionLag_Used				: LREAL;			
	{attribute 'tc_no_symbol'}                	                			
	_maxPositionLagTime_Used			: LREAL;	
	{attribute 'tc_no_symbol'}                	                					
	_softPositionLimitMaxActive_Used	: BOOL;				
	{attribute 'tc_no_symbol'}                	                			
	_softPositionLimitMinActive_Used	: BOOL;		
	{attribute 'tc_no_symbol'}                	                					
	_softPositionLimitMax_Used			: LREAL;	
	{attribute 'tc_no_symbol'}                	                					
	_softPositionLimitMin_Used			: LREAL;
	{attribute 'tc_no_symbol'}                	
	_MaxDriveOffDelay_Used				: DINT;
	{attribute 'tc_no_symbol'}   
	_HomeMode_Used						: INT;   
	_HomingCamSearchDirection_Used		: BOOL;  
	_HomingSyncSearchDirection_Used		: BOOL;               			
	_MaxDeceleration					: LREAL;
	{attribute 'tc_no_symbol'}                	                			
	_r_SetWrite_Trig					: ARRAY[0..10] OF R_TRIG;
	{attribute 'tc_no_symbol'}                	                			
	_r_SetRead_Trig						: ARRAY[0..10] OF R_TRIG;
	{attribute 'tc_no_symbol'}                	                			
	_r_Get_Trig							: R_TRIG;
	{attribute 'tc_no_symbol'}                	                			
	_CMD_ReadMaxDecelADS				: ADSREAD;
	{attribute 'tc_no_symbol'}                	                			
	_CMD_WriteParameterSet				: ARRAY[0..10] OF MC_WRITEPARAMETER;
	{attribute 'tc_no_symbol'}                	                			
	_CMD_ReadParameterSet				: ARRAY[0..10] OF MC_READPARAMETER;
	{attribute 'tc_no_symbol'}                	                			
	_CMD_ReadParameterGet				: ARRAY[0..10] OF MC_READPARAMETER;   
	{attribute 'tc_no_symbol'}   			
	_i									: USINT;
	{attribute 'tc_no_symbol'}                	                			
	_r_trig								: ARRAY[0..3] OF R_TRIG;
END_VAR
// Parameter Set
IF _Axis.Status.Disabled AND NOT Control.SystemTime.FirstCycle THEN
	
	//Set Torque Limits
	IF (_ManHome.Enabled OR _AutoHome) THEN
		_ServoTorqueLimit := F_CheckIndexBounds_UINT(10,100,_HomingTorqueLimit)*10;
	ELSE
		_ServoTorqueLimit := F_CheckIndexBounds_UINT(10,100,_NormalTorqueLimit)*10;
	END_IF;

	// Home Position Offset Value Set
	IF _Settings.HomeOffsetPosition <> _homeOffsetPosition_Used THEN
		_homeOffsetPosition_Used := _Settings.HomeOffsetPosition;
	END_IF
	
	// Maximum Position Lag Value Set
	_r_SetWrite_Trig[0](CLK:= _Settings.MaxPositionLag <> _maxPositionLag_Used);
	_CMD_WriteParameterSet[0](Axis := _Axis, Execute := _r_SetWrite_Trig[0].Q, ParameterNumber := MC_AxisParameter.MaxPositionLag,Value := _Settings.MaxPositionLag);
	_r_SetRead_Trig[0](CLK:= _CMD_WriteParameterSet[0].Done);
	_CMD_ReadParameterSet[0](Axis := _Axis, Enable := _r_SetRead_Trig[0].Q, ParameterNumber := MC_AxisParameter.MaxPositionLag,ReadMode := E_ReadMode.READMODE_ONCE);
	IF _CMD_ReadParameterSet[0].Valid THEN 
		_maxPositionLag_Used := _CMD_ReadParameterSet[0].Value; 
	END_IF

	// Maximum Position Lag Filter Time Set
	_r_SetWrite_Trig[1](CLK:=_Settings.MaxPositionLagTime <> _maxPositionLagTime_Used);
	_CMD_WriteParameterSet[1](Axis := _Axis, Execute := _r_SetWrite_Trig[1].Q, ParameterNumber := MC_AxisParameter.AxisMaxPosLagFilterTime, Value := _Settings.MaxPositionLagTime);
	_r_SetRead_Trig[1](CLK:= _CMD_WriteParameterSet[1].Done);
	_CMD_ReadParameterSet[1](Axis := _Axis, Enable := _r_SetRead_Trig[1].Q, ParameterNumber := MC_AxisParameter.AxisMaxPosLagFilterTime, ReadMode := E_ReadMode.READMODE_ONCE);
	IF _CMD_ReadParameterSet[1].Valid THEN 
		_maxPositionLagTime_Used := _CMD_ReadParameterSet[1].Value; 
	END_IF

	// Soft Position Limit Maximum Active Set
	_r_SetWrite_Trig[2](CLK:=_Settings.SoftPositionLimitMaxActive <> _softPositionLimitMaxActive_Used);
	_CMD_WriteParameterSet[2](Axis := _Axis, Execute := _r_SetWrite_Trig[2].Q, ParameterNumber := MC_AxisParameter.AxisEnMaxSoftPosLimit,Value := BOOL_TO_LREAL(_Settings.SoftPositionLimitMaxActive));
	_r_SetRead_Trig[2](CLK:= _CMD_WriteParameterSet[2].Done);
	_CMD_ReadParameterSet[2](Axis := _Axis, Enable := _r_SetRead_Trig[2].Q, ParameterNumber := MC_AxisParameter.AxisEnMaxSoftPosLimit, ReadMode := E_ReadMode.READMODE_ONCE);
	IF _CMD_ReadParameterSet[2].Valid THEN 
		_softPositionLimitMaxActive_Used := LREAL_TO_BOOL(_CMD_ReadParameterSet[2].Value); 
	END_IF
	
	// Soft Position Limit Minimum Active Set
	_r_SetWrite_Trig[3](CLK:=_Settings.SoftPositionLimitMinActive <> _softPositionLimitMinActive_Used);
	_CMD_WriteParameterSet[3](Axis := _Axis, Execute := _r_SetWrite_Trig[3].Q, ParameterNumber := MC_AxisParameter.AxisEnMinSoftPosLimit, Value := BOOL_TO_LREAL(_Settings.SoftPositionLimitMinActive));
	_r_SetRead_Trig[3](CLK:= _CMD_WriteParameterSet[3].Done);
	_CMD_ReadParameterSet[3](Axis := _Axis, Enable := _r_SetRead_Trig[3].Q, ParameterNumber := MC_AxisParameter.AxisEnMinSoftPosLimit, ReadMode := E_ReadMode.READMODE_ONCE);
	IF _CMD_ReadParameterSet[3].Valid THEN 
		_softPositionLimitMinActive_Used := LREAL_TO_BOOL(_CMD_ReadParameterSet[3].Value); 
	END_IF
	
	// Soft Position Limit Maximum Value Set
	_r_SetWrite_Trig[4](CLK:=_Settings.SoftPositionLimitMax <> _softPositionLimitMax_Used);
	_CMD_WriteParameterSet[4](Axis := _Axis, Execute := _r_SetWrite_Trig[4].Q, ParameterNumber := MC_AxisParameter.AxisMaxSoftPosLimit, Value := _Settings.SoftPositionLimitMax);
	_r_SetRead_Trig[4](CLK:=_CMD_WriteParameterSet[4].Done);
	_CMD_ReadParameterSet[4](Axis := _Axis, Enable := _r_SetRead_Trig[4].Q, ParameterNumber := MC_AxisParameter.AxisMaxSoftPosLimit, ReadMode := E_ReadMode.READMODE_ONCE);
	IF _CMD_ReadParameterSet[4].Valid THEN 
		_softPositionLimitMax_Used := _CMD_ReadParameterSet[4].Value; 
	END_IF
	
	// Soft Position Limit Minimum Value Set
	_r_SetWrite_Trig[5](CLK:=_Settings.SoftPositionLimitMin <> _softPositionLimitMin_Used);
	_CMD_WriteParameterSet[5](Axis := _Axis, Execute := _r_SetWrite_Trig[5].Q, ParameterNumber := MC_AxisParameter.AxisMinSoftPosLimit, Value := _Settings.SoftPositionLimitMin);
	_r_SetRead_Trig[5](CLK:=_CMD_WriteParameterSet[5].Done);
	_CMD_ReadParameterSet[5](Axis := _Axis, Enable := _r_SetRead_Trig[5].Q, ParameterNumber := MC_AxisParameter.AxisMinSoftPosLimit, ReadMode := E_ReadMode.READMODE_ONCE);
	IF _CMD_ReadParameterSet[5].Valid THEN 
		_softPositionLimitMin_Used := _CMD_ReadParameterSet[5].Value; 
	END_IF
	
	// Homing mode direction set - FALSE = FWD	
	CASE _HomeMode OF
		0: _Settings.HomingCamSearchDirection := TRUE; _Settings.HomingSyncSearchDirection := FALSE;
		1: _Settings.HomingCamSearchDirection := FALSE; _Settings.HomingSyncSearchDirection := FALSE;
		2: _Settings.HomingCamSearchDirection := FALSE; _Settings.HomingSyncSearchDirection := TRUE;
	END_CASE
	
	_r_SetWrite_Trig[6](CLK:=_Settings.HomingCamSearchDirection <> _HomingCamSearchDirection_Used);
	_CMD_WriteParameterSet[6](Axis := _Axis, Execute := _r_SetWrite_Trig[6].Q, ParameterNumber := MC_AxisParameter.AxisEncoderHomingInvDirCamSearch, Value := BOOL_TO_LREAL(_Settings.HomingCamSearchDirection));
	_r_SetRead_Trig[6](CLK:=_CMD_WriteParameterSet[6].Done);
	_CMD_ReadParameterSet[6](Axis := _Axis, Enable := _r_SetRead_Trig[6].Q, ParameterNumber := MC_AxisParameter.AxisEncoderHomingInvDirCamSearch, ReadMode := E_ReadMode.READMODE_ONCE);
	IF _CMD_ReadParameterSet[6].Valid THEN 
		_HomingCamSearchDirection_Used		:= LREAL_TO_BOOL(_CMD_ReadParameterSet[6].Value); 
	END_IF;
	
	_r_SetWrite_Trig[7](CLK:=_Settings.HomingSyncSearchDirection <> _HomingSyncSearchDirection_Used);
	_CMD_WriteParameterSet[7](Axis := _Axis, Execute := _r_SetWrite_Trig[6].Q, ParameterNumber := MC_AxisParameter.AxisEncoderHomingInvDirSyncSearch, Value := BOOL_TO_LREAL(_Settings.HomingSyncSearchDirection));
	_r_SetRead_Trig[7](CLK:=_CMD_WriteParameterSet[7].Done);
	_CMD_ReadParameterSet[7](Axis := _Axis, Enable := _r_SetRead_Trig[6].Q, ParameterNumber := MC_AxisParameter.AxisEncoderHomingInvDirSyncSearch, ReadMode := E_ReadMode.READMODE_ONCE);
	IF _CMD_ReadParameterSet[7].Valid THEN
		_HomingSyncSearchDirection_Used		:= LREAL_TO_BOOL(_CMD_ReadParameterSet[7].Value); 
	END_IF	
END_IF

// Parameter Get
_r_Get_Trig(CLK:= _UpdateDriveParameters OR Control.SystemTime.FirstCycle);

// Drive Status
_DriveStatus :=  F_ConvWordToSTAX5000DriveStatus(wDriveStatus:= _DriveStatusWord);

// Maximum Deceleration
_CMD_ReadMaxDecelADS(NETID := '',PORT := 501,IDXGRP := 16#00004002,IDXOFFS := 16#000000F2,LEN := 8,DESTADDR := ADR(_MaxDeceleration),READ := _r_Get_Trig.Q,TMOUT := ,BUSY => ,ERR => ,ERRID => ,);
_MaximumDeceleration := _MaxDeceleration;

// Maximum Position Lag Value Set
_CMD_ReadParameterGet[0](Axis := _Axis, Enable := _r_Get_Trig.Q, ParameterNumber := MC_AxisParameter.AxisMaxPosLagValue,ReadMode := E_ReadMode.READMODE_ONCE);
IF _CMD_ReadParameterGet[0].Valid THEN 
	_Settings.MaxPositionLag := _CMD_ReadParameterGet[0].Value; 
END_IF

// Maximum Position Lag Filter Time Get
_CMD_ReadParameterGet[1](Axis := _Axis, Enable := _r_Get_Trig.Q, ParameterNumber := MC_AxisParameter.AxisMaxPosLagFilterTime,ReadMode := E_ReadMode.READMODE_ONCE);
IF _CMD_ReadParameterGet[1].Valid THEN 
	_Settings.MaxPositionLagTime := _CMD_ReadParameterGet[1].Value; 
END_IF

// Soft Position Limit Maximum Active Get
_CMD_ReadParameterGet[2](Axis := _Axis, Enable := _r_Get_Trig.Q, ParameterNumber := MC_AxisParameter.AxisEnMaxSoftPosLimit,ReadMode := E_ReadMode.READMODE_ONCE);
IF _CMD_ReadParameterGet[2].Valid THEN 
	_Settings.SoftPositionLimitMaxActive := LREAL_TO_BOOL(_CMD_ReadParameterGet[2].Value); 
END_IF

// Soft Position Limit Minimum Active Get
_CMD_ReadParameterGet[3](Axis := _Axis, Enable := _r_Get_Trig.Q, ParameterNumber := MC_AxisParameter.AxisEnMinSoftPosLimit,ReadMode := E_ReadMode.READMODE_ONCE);
IF _CMD_ReadParameterGet[3].Valid THEN 
	_Settings.SoftPositionLimitMinActive := LREAL_TO_BOOL(_CMD_ReadParameterGet[3].Value); 
END_IF

// Soft Position Limit Maximum Value Get
_CMD_ReadParameterGet[4](Axis := _Axis, Enable := _r_Get_Trig.Q, ParameterNumber := MC_AxisParameter.AxisMaxSoftPosLimit,ReadMode := E_ReadMode.READMODE_ONCE);
IF _CMD_ReadParameterGet[4].Valid THEN 
	_Settings.SoftPositionLimitMax := _CMD_ReadParameterGet[4].Value; 
END_IF

// Soft Position Limit Minimum Value Get
_CMD_ReadParameterGet[5](Axis := _Axis, Enable := _r_Get_Trig.Q, ParameterNumber := MC_AxisParameter.AxisMinSoftPosLimit,ReadMode := E_ReadMode.READMODE_ONCE);
IF _CMD_ReadParameterGet[5].Valid THEN 
	_Settings.SoftPositionLimitMin := _CMD_ReadParameterGet[5].Value; 
END_IF

// Modulo Factor Value Get
_CMD_ReadParameterGet[6](Axis := _Axis, Enable := _r_Get_Trig.Q, ParameterNumber := MC_AxisParameter.AxisEncoderModuloValue,ReadMode := E_ReadMode.READMODE_ONCE);
IF _CMD_ReadParameterGet[6].Valid THEN 
	_Settings.ModuloFactor := _CMD_ReadParameterGet[6].Value; 
END_IF

//Check for Function Block Errors
_r_trig[0](CLK:=_CMD_ReadMaxDecelADS.ERR);	
IF _r_trig[0].Q THEN _AlarmNum := _CMD_ReadMaxDecelADS.ERRID; END_IF

FOR _i := 0 TO 10 BY 1 DO
 	_r_trig[1](CLK:=_CMD_WriteParameterSet[_i].Error);	
	IF _r_trig[1].Q THEN _AlarmNum := _CMD_WriteParameterSet[_i].ErrorID;END_IF
	_r_trig[2](CLK:=_CMD_ReadParameterSet[_i].Error);	
	IF _r_trig[2].Q THEN _AlarmNum := _CMD_ReadParameterSet[_i].ErrorID;END_IF
    _r_trig[3](CLK:=_CMD_ReadParameterGet[_i].Error);
	IF _r_trig[3].Q THEN _AlarmNum := _CMD_ReadParameterGet[_i].ErrorID;END_IF
END_FOR
END_METHOD

METHOD PRIVATE M_StateControl
VAR_INPUT
END_VAR
VAR_INST
	{attribute 'tc_no_symbol'}                	                			
	_StepTimerET						: REAL;
	{attribute 'tc_no_symbol'}                	                			
	_StepTimerPT						: ARRAY[0..20] OF REAL;
	{attribute 'tc_no_symbol'}                	                			
	_StepTimerDN						: BOOL;
	{attribute 'tc_no_symbol'}                	                			
	_last_Step							: DINT;					

END_VAR
VAR_INST // added by the converter: edge detectors and wires of the graphical bodies
    _w1 : BOOL;
END_VAR
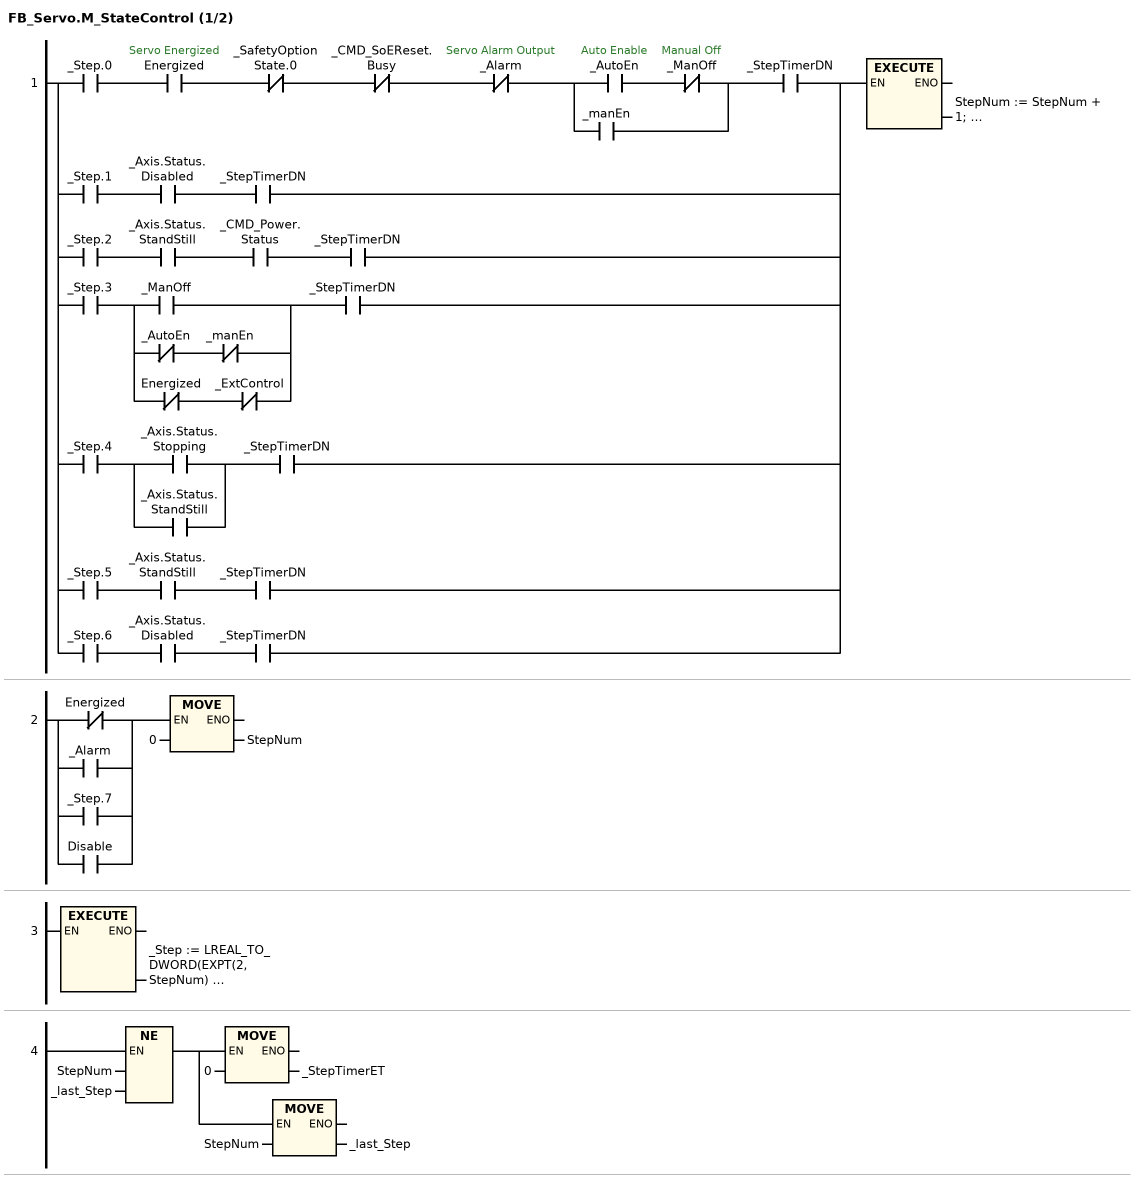
// NETWORK 1
//   Energized: Servo Energized
//   _Alarm: Servo Alarm Output
//   _AutoEn: Auto Enable
//   _ManOff: Manual Off
IF _Step.0 AND Energized AND NOT _SafetyOptionState.0 AND NOT _CMD_SoEReset.Busy AND NOT _Alarm AND (_AutoEn AND NOT _ManOff OR _manEn) AND _StepTimerDN OR _Step.1 AND _Axis.Status.Disabled AND _StepTimerDN OR _Step.2 AND _Axis.Status.StandStill AND _CMD_Power.Status AND _StepTimerDN OR _Step.3 AND (_ManOff OR NOT _AutoEn AND NOT _manEn OR NOT Energized AND NOT _ExtControl) AND _StepTimerDN OR _Step.4 AND (_Axis.Status.Stopping OR _Axis.Status.StandStill) AND _StepTimerDN OR _Step.5 AND _Axis.Status.StandStill AND _StepTimerDN OR _Step.6 AND _Axis.Status.Disabled AND _StepTimerDN THEN
    StepNum := StepNum + 1;
END_IF

// NETWORK 2
//   StepNum: Servo State Control Step Number Output
IF NOT Energized OR _Alarm OR _Step.7 OR Disable THEN StepNum := 0; END_IF

// NETWORK 3
_Step := LREAL_TO_DWORD(EXPT(2, StepNum));

// NETWORK 4
//   StepNum: Servo State Control Step Number Output
_w1 := StepNum <> _last_Step;
IF _w1 THEN _StepTimerET := 0; END_IF
IF _w1 THEN _last_Step := StepNum; END_IF

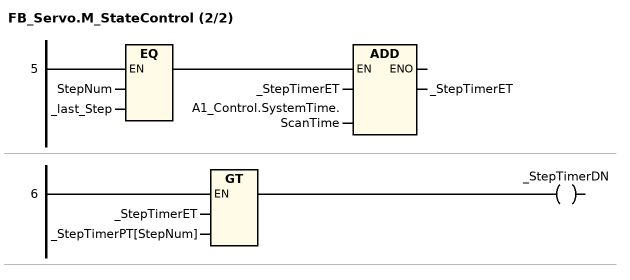
// NETWORK 5
//   StepNum: Servo State Control Step Number Output
//   A1_Control.SystemTime.ScanTime: Last scan time (Seconds)
IF StepNum = _last_Step THEN _StepTimerET := _StepTimerET + A1_Control.SystemTime.ScanTime; END_IF

// NETWORK 6
_StepTimerDN := _StepTimerET > _StepTimerPT[StepNum];
END_METHOD

METHOD PRIVATE M_StateOutputs
VAR_INPUT
END_VAR
VAR_INST
	{attribute 'tc_no_symbol'}                	                			
	_power				: BOOL;
	{attribute 'tc_no_symbol'}                	                			
	_decelRate			: LREAL;
	{attribute 'tc_no_symbol'}                	                			
	_CMD_Reset			: MC_RESET;
	{attribute 'tc_no_symbol'}                	                			
	_CMD_Stop			: MC_STOP;
END_VAR
VAR_INST // added by the converter: edge detectors and wires of the graphical bodies
    _rt1, _rt2, _rt3, _rt4 : R_TRIG;
    _w1 : BOOL;
END_VAR
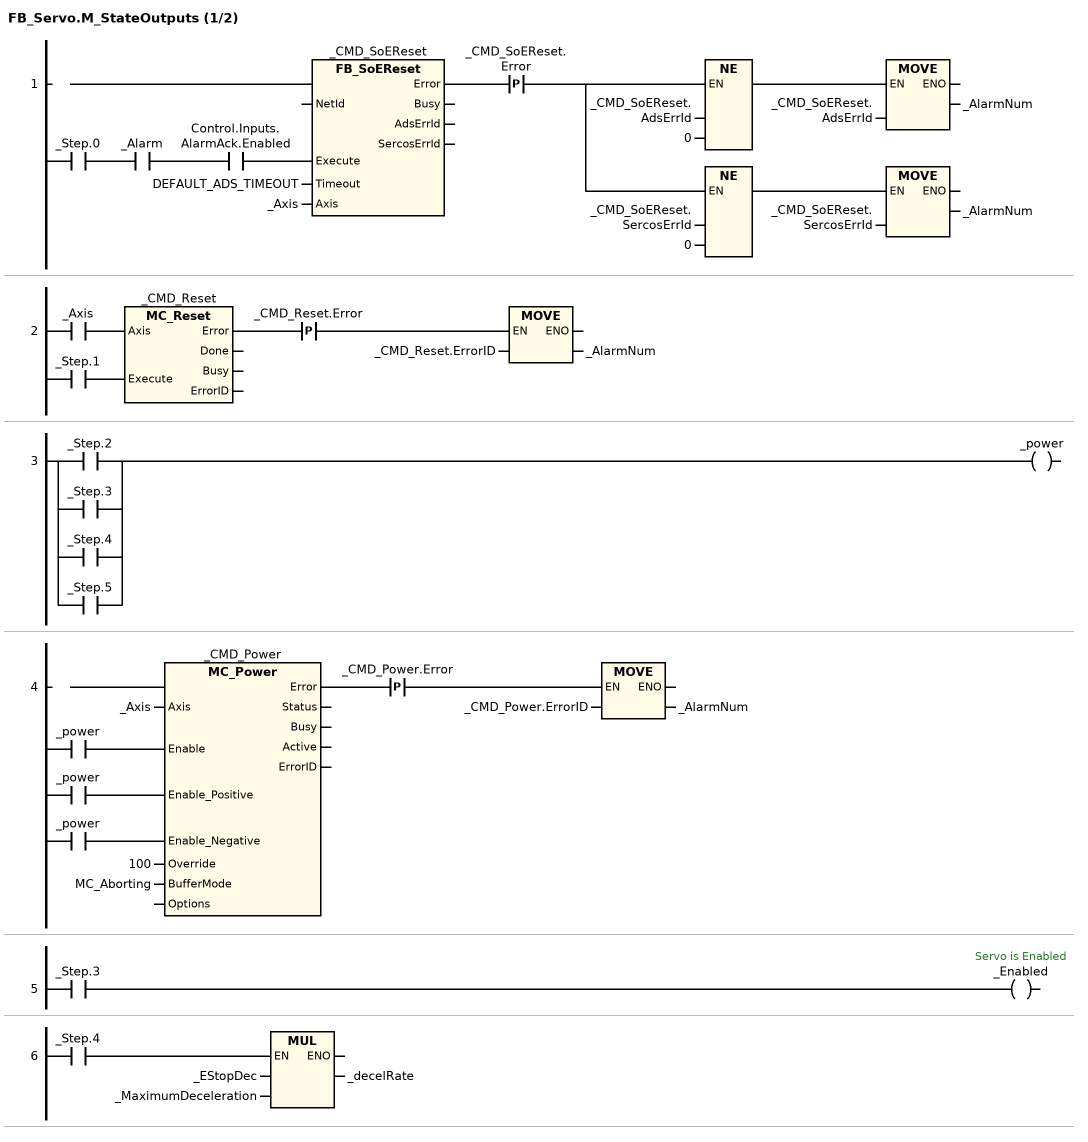
// NETWORK 1
_CMD_SoEReset(
    Execute := _Step.0 AND _Alarm AND Control.Inputs.AlarmAck.Enabled,
    Timeout := DEFAULT_ADS_TIMEOUT,
    Axis := _Axis); // FB_SoEReset
_rt1(CLK := _CMD_SoEReset.Error);
_w1 := _CMD_SoEReset.Error AND _rt1.Q;
IF _w1 AND _CMD_SoEReset.AdsErrId <> 0 THEN _AlarmNum := _CMD_SoEReset.AdsErrId; END_IF
IF _w1 AND _CMD_SoEReset.SercosErrId <> 0 THEN _AlarmNum := _CMD_SoEReset.SercosErrId; END_IF

// NETWORK 2
_CMD_Reset(Axis := _Axis, Execute := _Step.1); // MC_Reset
_rt2(CLK := _CMD_Reset.Error);
IF _CMD_Reset.Error AND _rt2.Q THEN _AlarmNum := _CMD_Reset.ErrorID; END_IF

// NETWORK 3
_power := _Step.2 OR _Step.3 OR _Step.4 OR _Step.5;

// NETWORK 4
_CMD_Power(
    Axis := _Axis,
    Enable := _power,
    Enable_Positive := _power,
    Enable_Negative := _power,
    Override := 100,
    BufferMode := MC_Aborting); // MC_Power
_rt3(CLK := _CMD_Power.Error);
IF _CMD_Power.Error AND _rt3.Q THEN _AlarmNum := _CMD_Power.ErrorID; END_IF

// NETWORK 5
//   _Enabled: Servo is Enabled
_Enabled := _Step.3;

// NETWORK 6
//   _EStopDec: EStop Deceleration Percentage
//   _MaximumDeceleration: Maximum Deceleration of the System
IF _Step.4 THEN _decelRate := _EStopDec * _MaximumDeceleration; END_IF

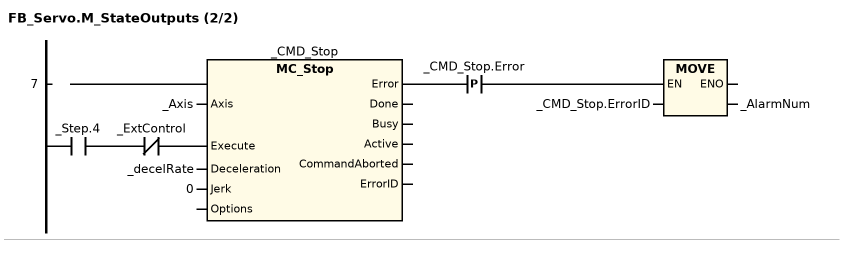
// NETWORK 7
_CMD_Stop(Axis := _Axis, Execute := _Step.4 AND NOT _ExtControl, Deceleration := _decelRate, Jerk := 0); // MC_Stop
_rt4(CLK := _CMD_Stop.Error);
IF _CMD_Stop.Error AND _rt4.Q THEN _AlarmNum := _CMD_Stop.ErrorID; END_IF
END_METHOD

METHOD PRIVATE M_UnlatchManuals
VAR_INPUT
END_VAR
VAR_INST
END_VAR
VAR_INST // added by the converter: edge detectors and wires of the graphical bodies
    _rt1, _rt2, _rt3, _rt4, _rt5 : R_TRIG;
END_VAR
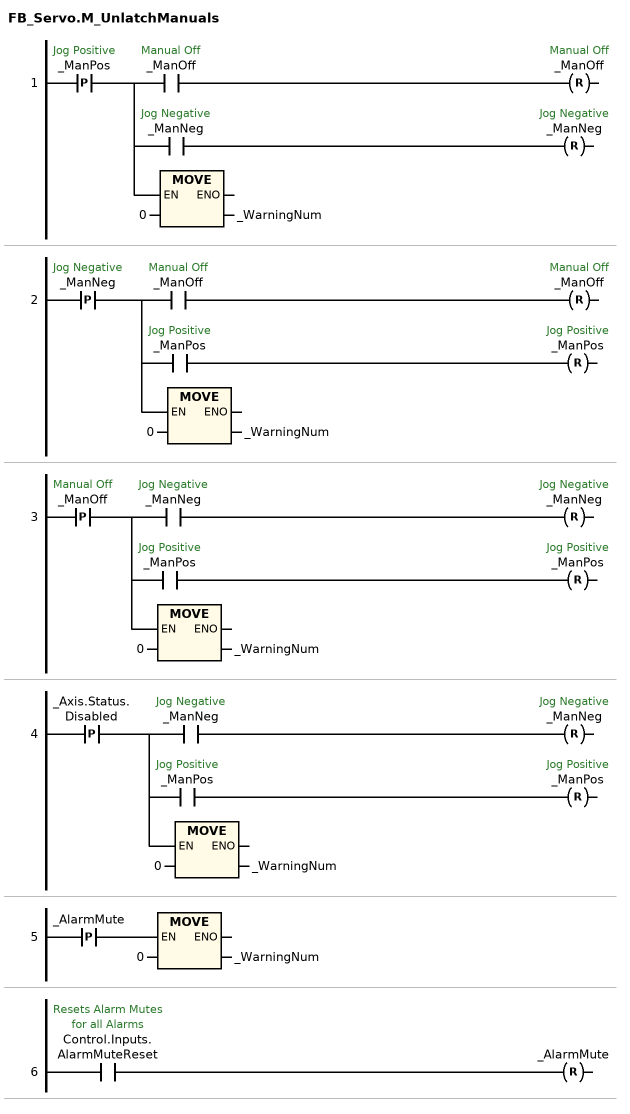
// NETWORK 1
//   _ManPos: Jog Positive
//   _ManOff: Manual Off
//   _ManNeg: Jog Negative
_rt1(CLK := _ManPos);
_ManOff R= _rt1.Q AND _ManOff;
_ManNeg R= _rt1.Q AND _ManNeg;
IF _rt1.Q THEN _WarningNum := 0; END_IF

// NETWORK 2
//   _ManNeg: Jog Negative
//   _ManOff: Manual Off
//   _ManPos: Jog Positive
_rt2(CLK := _ManNeg);
_ManOff R= _rt2.Q AND _ManOff;
_ManPos R= _rt2.Q AND _ManPos;
IF _rt2.Q THEN _WarningNum := 0; END_IF

// NETWORK 3
//   _ManOff: Manual Off
//   _ManNeg: Jog Negative
//   _ManPos: Jog Positive
_rt3(CLK := _ManOff);
_ManNeg R= _rt3.Q AND _ManNeg;
_ManPos R= _rt3.Q AND _ManPos;
IF _rt3.Q THEN _WarningNum := 0; END_IF

// NETWORK 4
//   _ManNeg: Jog Negative
//   _ManPos: Jog Positive
_rt4(CLK := _Axis.Status.Disabled);
_ManNeg R= _rt4.Q AND _ManNeg;
_ManPos R= _rt4.Q AND _ManPos;
IF _rt4.Q THEN _WarningNum := 0; END_IF

// NETWORK 5
_rt5(CLK := _AlarmMute);
IF _rt5.Q THEN _WarningNum := 0; END_IF

// NETWORK 6
//   Control.Inputs.AlarmMuteReset: Resets Alarm Mutes for all Alarms
_AlarmMute R= Control.Inputs.AlarmMuteReset;
END_METHOD

METHOD PRIVATE M_WarningMonitor
VAR_INPUT
END_VAR
VAR_INST
	{attribute 'tc_no_symbol'}                	                			
	_R_Trig				:   ARRAY[0..2] OF R_TRIG;
END_VAR
VAR_INST // added by the converter: edge detectors and wires of the graphical bodies
    _w1, _w2 : BOOL;
END_VAR
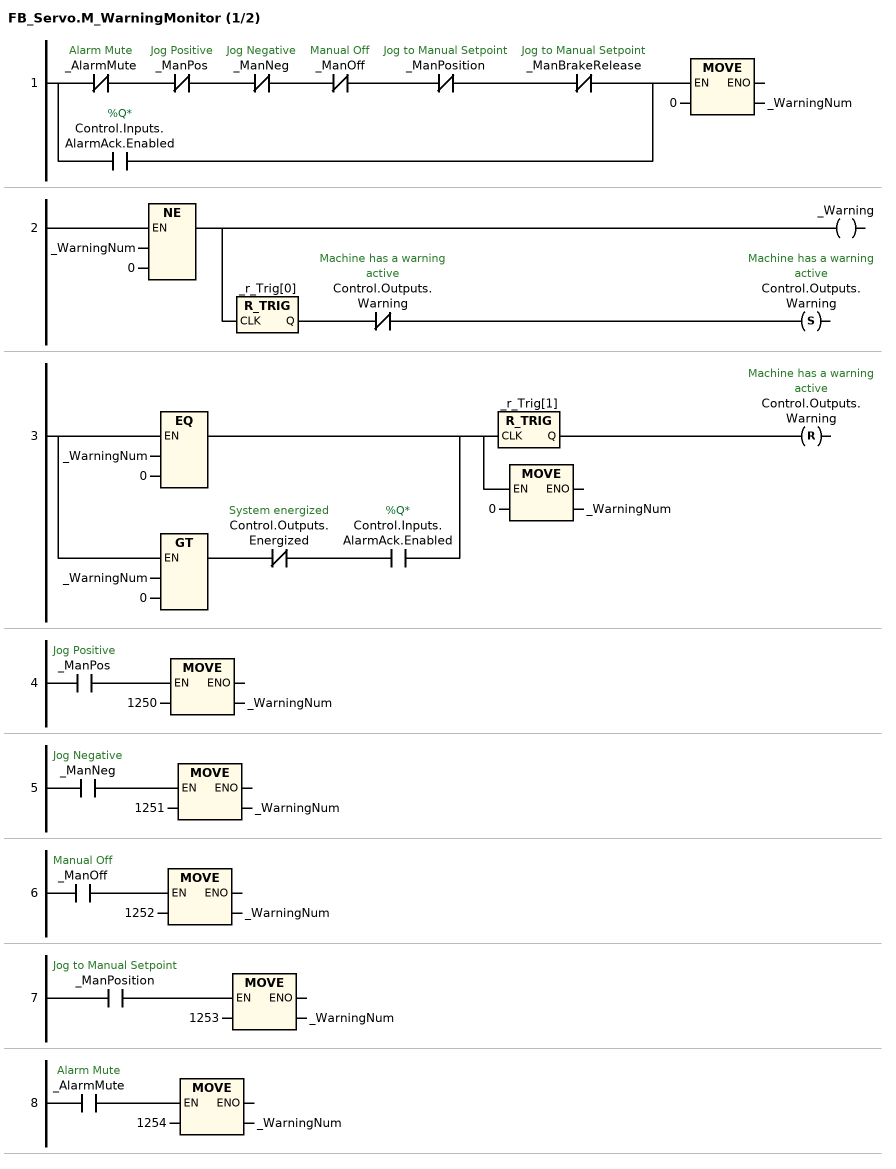
// NETWORK 1
//   _AlarmMute: Alarm Mute
//   _ManPos: Jog Positive
//   _ManNeg: Jog Negative
//   _ManOff: Manual Off
//   _ManPosition: Jog to Manual Setpoint
//   _ManBrakeRelease: Jog to Manual Setpoint
//   Control.Inputs.AlarmAck.Enabled: AT %Q*
IF NOT _AlarmMute AND NOT _ManPos AND NOT _ManNeg AND NOT _ManOff AND NOT _ManPosition AND NOT _ManBrakeRelease OR Control.Inputs.AlarmAck.Enabled THEN
    _WarningNum := 0;
END_IF

// NETWORK 2
//   Control.Outputs.Warning: Machine has a warning active
_w1 := _WarningNum <> 0;
_Warning := _w1;
_r_Trig[0](CLK := _w1); // R_TRIG
Control.Outputs.Warning S= _r_Trig[0].Q AND NOT Control.Outputs.Warning;

// NETWORK 3
//   Control.Outputs.Energized: System energized
//   Control.Inputs.AlarmAck.Enabled: AT %Q*
//   Control.Outputs.Warning: Machine has a warning active
_w2 := _WarningNum = 0 OR _WarningNum > 0 AND NOT Control.Outputs.Energized AND Control.Inputs.AlarmAck.Enabled;
_r_Trig[1](CLK := _w2); // R_TRIG
Control.Outputs.Warning R= _r_Trig[1].Q;
IF _w2 THEN _WarningNum := 0; END_IF

// NETWORK 4
//   _ManPos: Jog Positive
IF _ManPos THEN _WarningNum := 1250; END_IF

// NETWORK 5
//   _ManNeg: Jog Negative
IF _ManNeg THEN _WarningNum := 1251; END_IF

// NETWORK 6
//   _ManOff: Manual Off
IF _ManOff THEN _WarningNum := 1252; END_IF

// NETWORK 7
//   _ManPosition: Jog to Manual Setpoint
IF _ManPosition THEN _WarningNum := 1253; END_IF

// NETWORK 8
//   _AlarmMute: Alarm Mute
IF _AlarmMute THEN _WarningNum := 1254; END_IF

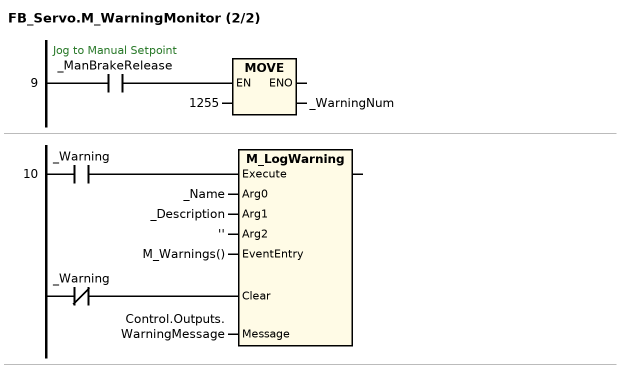
// NETWORK 9
//   _ManBrakeRelease: Jog to Manual Setpoint
IF _ManBrakeRelease THEN _WarningNum := 1255; END_IF

// NETWORK 10
M_LogWarning(Execute := _Warning, Arg0 := _Name, Arg1 := _Description, Arg2 := '', EventEntry := M_Warnings(), Clear := NOT _Warning, Message := Control.Outputs.WarningMessage);
END_METHOD

METHOD PRIVATE M_Warnings : TcEventEntry
VAR_INPUT
END_VAR
VAR_INST
END_VAR
CASE _WarningNum OF	
1150:    M_Warnings := 	TC_Events.TcServo.W_1150;			
1151:    M_Warnings :=  TC_Events.TcServo.W_1151;			
1152:    M_Warnings := 	TC_Events.TcServo.W_1152;			
1153:    M_Warnings := 	TC_Events.TcServo.W_1153;			
1154:    M_Warnings := 	TC_Events.TcServo.W_1154;	
1155:    M_Warnings :=  TC_Events.TcServo.W_1155;	
ELSE
		 M_Warnings := 	TC_Events.TcServo.W_Undefined;
END_CASE
END_METHOD

{attribute 'monitoring' := 'variable'}
PROPERTY PUBLIC ManBrakeRelease : Bool
SET
_ManBrakeRelease := ManBrakeRelease;
END_SET
END_PROPERTY

{attribute 'monitoring' := 'variable'}
PROPERTY PUBLIC ManEn : Bool
GET
ManEn := _ManEn;
END_GET
SET
_ManEn := ManEn;
END_SET
END_PROPERTY

{attribute 'monitoring' := 'variable'}
PROPERTY PUBLIC ManHome : REFERENCE TO ST_Selection
GET
ManHome REF= _ManHome;
END_GET
SET
_ManHome := ManHome;
END_SET
END_PROPERTY

{attribute 'monitoring' := 'variable'}
PROPERTY PUBLIC MoveDynamic : REFERENCE TO ARRAY[1..4] OF BOOL
GET // PUBLIC
MoveDynamic REF= _MoveDynamic;
END_GET
SET
_MoveDynamic := MoveDynamic;
END_SET
END_PROPERTY

{attribute 'monitoring' := 'variable'}
PROPERTY PUBLIC MovePos : REFERENCE TO ARRAY[1..4] OF BOOL
GET // PUBLIC
MovePos REF= _MovePos;
END_GET
SET
_MovePos := MovePos;
END_SET
END_PROPERTY

{attribute 'monitoring' := 'variable'}
PROPERTY PUBLIC MovePosSync : Bool
SET
_MovePosSync := MovePosSync;
END_SET
END_PROPERTY

{attribute 'monitoring' := 'variable'}
PROPERTY PUBLIC MoveSuperImpose : Bool
SET
_MoveSuperImpose := MoveSuperImpose;
END_SET
END_PROPERTY

{attribute 'monitoring' := 'variable'}
PROPERTY PUBLIC Moving : Bool
GET
Moving := _Moving;
END_GET
END_PROPERTY

{attribute 'monitoring' := 'variable'}
PROPERTY PUBLIC Name : String[15]
GET
Name := _Name;
END_GET
SET
_Name := Name;
END_SET
END_PROPERTY

{attribute 'monitoring' := 'variable'}
PROPERTY PUBLIC PosDynamicOK : REFERENCE TO ARRAY[1..4] OF BOOL
GET // PUBLIC
PosDynamicOK REF= _PosDynamicOK;
END_GET
END_PROPERTY

{attribute 'Suspress_wrn_C0410'}
PROPERTY PUBLIC PosMove : REFERENCE TO ARRAY[1..4] OF ST_MovePosition_SP
GET // PUBLIC
Posmove REF= _PosMove;
END_GET
SET
_Posmove := PosMove;
END_SET
END_PROPERTY

{attribute 'monitoring' := 'variable'}
PROPERTY PUBLIC PosMoveHome : REFERENCE TO ST_HomePosition_SP;
GET // PUBLIC
PosMoveHome REF= _PosMoveHome;
END_GET
SET
_PosMoveHome := PosMoveHome;
END_SET
END_PROPERTY

{attribute 'monitoring' := 'variable'}
PROPERTY PUBLIC PosOK : REFERENCE TO ARRAY[1..4] OF BOOL
GET // PUBLIC
PosOK REF= _PosOK;
END_GET
END_PROPERTY

{attribute 'monitoring' := 'variable'}
PROPERTY PUBLIC PosSyncOK : Bool
GET
PosSyncOK := _PosSyncOK;
END_GET
END_PROPERTY

{attribute 'monitoring' := 'variable'}
PROPERTY PUBLIC RunCam : Bool
SET
_RunCam := RunCam;
END_SET
END_PROPERTY

{attribute 'monitoring' := 'variable'}
PROPERTY PUBLIC StandStill : Bool
GET
StandStill := _StandStill;
END_GET
END_PROPERTY

{attribute 'monitoring' := 'variable'}
PROPERTY PUBLIC Unit : String[8]
GET
Unit := _Unit;
END_GET
SET
_Unit := Unit;
END_SET
END_PROPERTY

PROPERTY PUBLIC Variables : REFERENCE TO ARRAY[0..9] OF ST_Variable
GET
Variables REF= _Variables;
END_GET
END_PROPERTY

{attribute 'monitoring' := 'variable'}
PROPERTY PUBLIC Warning : Bool
GET
Warning := _Warning;
END_GET
END_PROPERTY

END_FUNCTION_BLOCK

(* stored: Version 1.1.0.1, ProductVersion 3.1.4024.3
   POU FB_Servo: Id {16cb79a1-c076-4a59-831f-2c230a7ff183}, SpecialFunc None
   Property Alarm: Id {51243af3-c8bd-4b19-9b53-f293f80cf333}
   Get Get: Id {cf64cd82-9032-46a4-b346-1a8658c0c1c6}
   Property AlarmMute: Id {2fe0601b-c58b-4900-bfdc-4823bbe53f51}
   Set Set: Id {431027cb-d30b-421b-9c67-e5de2ca21a40}
   Property AutoEn: Id {c79c3b75-bb6f-42a5-8922-dd72e70501ac}
   Get Get: Id {b52e2d04-f4ac-4659-8801-e833b236e3ca}
   Set Set: Id {f837c46e-226c-44a6-b093-cb547e92a86c}
   Property AutoHome: Id {92c63411-5401-4c1b-abf8-02d5b1e42759}
   Get Get: Id {3c005933-f776-4ac2-9827-0e8a6114bdc3}
   Set Set: Id {4b7662b4-fb19-4c87-8a85-6188525f8ed3}
   Property AxisEnabled: Id {74ca12b4-3bd3-4eb6-9c44-c83d92d47588}
   Get Get: Id {5b94e87b-090a-4fc5-886d-ec65a21b62b7}
   Property CamInSync: Id {b9cc822e-22c8-46b1-819f-87ac4c47cf50}
   Get Get: Id {9f09a8d6-e7ef-4f07-a5ac-9d54a38b87b8}
   Property ContinuousRun: Id {ad026966-3274-4b4c-b601-ef725a52b335}
   Get Get: Id {ccb74f09-2944-4781-9c90-b4db299d7f0b}
   Set Set: Id {d743d097-426b-4154-9320-db7945a1b49c}
   Property ContRun: Id {b71b8a62-8c56-4f71-a5e9-a62fff439d81}
   Set Set: Id {ec74b2fc-3c14-44fc-88d8-6bd5d3919612}
   Property Description: Id {fc78563d-3b2d-48b8-8144-c11ea4e2fc1c}
   Get Get: Id {25a9c31c-05aa-4b18-8bc3-bbf1bb25f8b9}
   Set Set: Id {cb8e16dd-8079-4f0a-837e-b063cba1a321}
   Property DigitalInputs: Id {ba9d062d-6a07-4fc8-aba0-0634989eb082}
   Get Get: Id {a43f2819-6296-4af6-b8ad-b81a6c43f5f8}
   Set Set: Id {b3e97a3c-c5a2-47fc-a13a-d6e19d51abd2}
   Property ExtControl: Id {efbd9c10-7bd6-42d5-b40f-b5049dd10df8}
   Set Set: Id {5f143108-50e2-4f77-9061-113aada9a81a}
   Property ExtManEn: Id {3c506b2a-bcd1-4f7d-bd60-06689a0675fc}
   Set Set: Id {95f60099-4224-4c52-89fe-984e542f6dad}
   Property Fault: Id {e17d4624-efe0-4e43-a27d-22579129b887}
   Set Set: Id {b63a8ec6-9e23-45cd-8889-486ab6d4466f}
   Property FaultTimer_ET: Id {ce3ff983-5eb8-4dc1-b5f7-2f970e66ca4e}
   Get Get: Id {56e43775-4a54-4d2e-9b90-2fabf444bc6d}
   Property FaultTimer_PT: Id {b643fc30-d94d-439b-a380-a2c56de28697}
   Get Get: Id {c06d368d-bcbc-4dcd-86d5-92a2c8f19395}
   Set Set: Id {9806af60-2f05-4658-aab8-4be7f9466579}
   Property ForceNeg: Id {bbc73d8a-1c8a-44f2-9fb4-407ecaf287a0}
   Get Get: Id {d8f92dbf-a39d-4565-9b23-0c4a5af9ca0b}
   Set Set: Id {117ac04c-0a4c-4cd6-965b-ff597a8c643e}
   Property ForcePos: Id {d3baabfc-3277-4ff9-926f-0f90e298baf1}
   Get Get: Id {f8b1b7f6-5ae8-40f2-8cef-0e40b62cc304}
   Set Set: Id {14dd8115-41a6-4ae7-a68b-9bc84eea4547}
   Property Homed: Id {82fb4980-bd58-44a0-b056-61923d785a13}
   Get Get: Id {272ca7ea-d8c4-4808-a812-da5f0e20c2f7}
   Property HomeMode: Id {5a17d1a9-3740-40b6-86b4-6115581f83e7}
   Get Get: Id {7b08f475-0517-48c3-9e7e-903a92bf822c}
   Set Set: Id {75e5c68c-9919-4c63-8a2c-be5cdad9ae83}
   Property Jog: Id {4ae3c193-1594-47de-a611-d60a8e0cb68a}
   Get Get: Id {37befdbb-5fe5-41c6-acd9-a95d81e3a96e}
   Set Set: Id {43af12d2-08d6-4262-9808-9052634b475d}
   Method M_AlarmMonitor: Id {4ec36063-b488-4071-ad8a-0e3556b07f18}
   Method M_Alarms: Id {5ea9ab63-8374-4bb3-8eb6-8a9b1e224fc9}
   Method M_BrakeControl: Id {7eb22851-e108-454c-a6e6-835368b9d7e2}
   Method M_ContinuousRun: Id {ce135928-5a90-479b-a3ea-37980bc79f68}
   Method M_ControlOutputs: Id {41eca18e-81fc-495e-b855-94959ce1fb83}
   Method M_Errors: Id {f78901b1-23b0-48cc-853a-850f8daa09e8}
   Method M_GetDiagnosis: Id {6a1ff3f6-9af3-4592-a17f-f90000b8e0e1}
   Method M_Homing: Id {e8f59e10-8be6-4f00-9775-bb68ed86d050}
   Method M_Jogging: Id {1ca8c097-9a69-4364-8506-42e3db2d0590}
   Method M_MotionDynamicMove: Id {8e8f348d-97f6-44e4-acc5-50f64a84fb81}
   Method M_MoveSuperImposed: Id {af1fd278-0e58-4954-8c87-48fee3b20af4}
   Method M_MoveToPosition: Id {fe94e7c9-b573-4e48-a5aa-6f0821c097b3}
   Method M_SettingsControl: Id {fb67c05d-e9de-426f-85cf-95d23d2abc89}
   Method M_StateControl: Id {35764898-bea9-4742-aec6-c7137e445d5e}
   Method M_StateOutputs: Id {279b5250-19db-4b4e-9301-9c510250a627}
   Method M_UnlatchManuals: Id {18fa7697-bb45-4278-a26b-b391ce6e2092}
   Method M_WarningMonitor: Id {d2bf7150-566d-4d47-9572-cfcf287cf358}
   Method M_Warnings: Id {b60aa26a-9b64-4e2a-a8e1-64f6ef044e42}
   Property ManBrakeRelease: Id {dd3785bd-b1be-4150-89a2-79ad3e03c64c}
   Set Set: Id {8f73f691-4025-484b-9373-2800e581fa94}
   Property ManEn: Id {647a5f82-0739-4816-8693-b41faec39e0d}
   Get Get: Id {339e45a0-237f-4aa3-8e3b-7dcc9486c317}
   Set Set: Id {81973c10-e0e9-4241-877e-facf89a40f15}
   Property ManHome: Id {c9c2a71b-ad2b-49ff-bff2-9b4f0f16d53e}
   Get Get: Id {ccf2b8d5-ff23-46cf-b904-8e6d31a51122}
   Set Set: Id {70712a77-64ef-4a45-8336-f334f3d3b0d1}
   Property MoveDynamic: Id {4158b0d2-5b91-4cac-ad1a-7e70dcd2b1a9}
   Get Get: Id {13786e9f-00af-4793-b7a8-eabded72ecb0}
   Set Set: Id {30e18da5-0ee8-4df1-b152-ef7e6685236a}
   Property MovePos: Id {4f73325f-350d-4029-8f4f-b9a2a5cbf1eb}
   Get Get: Id {ea75a7d4-aa18-41df-a495-6e2704468d00}
   Set Set: Id {68eff27f-639c-4b07-b453-f37123adbeea}
   Property MovePosSync: Id {f440f3ea-3e1b-49a5-9ce8-5e0983d39dbc}
   Set Set: Id {1e33ce11-f199-406b-a83c-9c95ae5a89ee}
   Property MoveSuperImpose: Id {87a0788c-fc61-4fc3-97b5-0333c184edc6}
   Set Set: Id {5c08faa4-8cf5-4cd5-bf92-749f22f2f909}
   Property Moving: Id {890e1b9b-5260-48d7-8e84-f362176c1f94}
   Get Get: Id {816a3b91-e04d-4af9-8baf-3f9a1710773c}
   Property Name: Id {9c420f1f-a8db-4033-8d2c-612c53ead349}
   Get Get: Id {6933fc74-66fe-4962-8209-6544f699a99d}
   Set Set: Id {c72c4432-acbf-4a81-a24f-bebf9706e306}
   Property PosDynamicOK: Id {898e614e-ad8e-45e2-97a9-3688452db53d}
   Get Get: Id {65b2cf78-fc68-4c1e-b9bf-876b04d21bd1}
   Property PosMove: Id {b82a1524-8f9d-4470-8fdc-d59841fcc3e8}
   Get Get: Id {5c3b1940-7106-497b-a011-6f16544a0c32}
   Set Set: Id {a4e297d9-7f4e-4a6c-9e04-f4ebf406bcee}
   Property PosMoveHome: Id {26a4d39f-7535-4932-b9df-a1264bcfe2c4}
   Get Get: Id {e87f6933-e8d8-4b07-a598-93aea9be4106}
   Set Set: Id {3187b9d1-6af0-4bdd-95f1-76ddcce9493c}
   Property PosOK: Id {fc087c67-f482-4ee1-aa38-4eb4ddeec320}
   Get Get: Id {ffc49613-fcab-4700-86cb-ec4dae451937}
   Property PosSyncOK: Id {61eedc8f-1f62-4dec-9705-66395dd285db}
   Get Get: Id {ba600b33-c068-47bf-9bc3-34db8cc89d38}
   Property RunCam: Id {223b22ee-810a-4f4a-a336-15ba297db390}
   Set Set: Id {cd29da64-65a9-44a5-94e7-e81da8bd8cd4}
   Property StandStill: Id {75608dd8-e64a-41a5-b4c8-09f7205f3148}
   Get Get: Id {09d3190e-fcf4-4233-bd98-7de1bd6200a8}
   Property Unit: Id {53a4cdd7-8493-4fd4-a0cf-41bdc4252480}
   Get Get: Id {716a23ee-4548-4d52-a9d3-3a31cd6c565e}
   Set Set: Id {d6efdcec-0007-4d3e-8d1e-9589405d6263}
   Property Variables: Id {dc5e2090-15fe-469c-94cd-a19ba9d8afec}
   Get Get: Id {15ef582a-c486-4c65-bf55-451eff0c0f3a}
   Property Warning: Id {e9c6e2c8-294f-48c6-b3d4-f9a17d32982d}
   Get Get: Id {e6417af1-1595-4f52-9f2c-fc4275143391} *)
